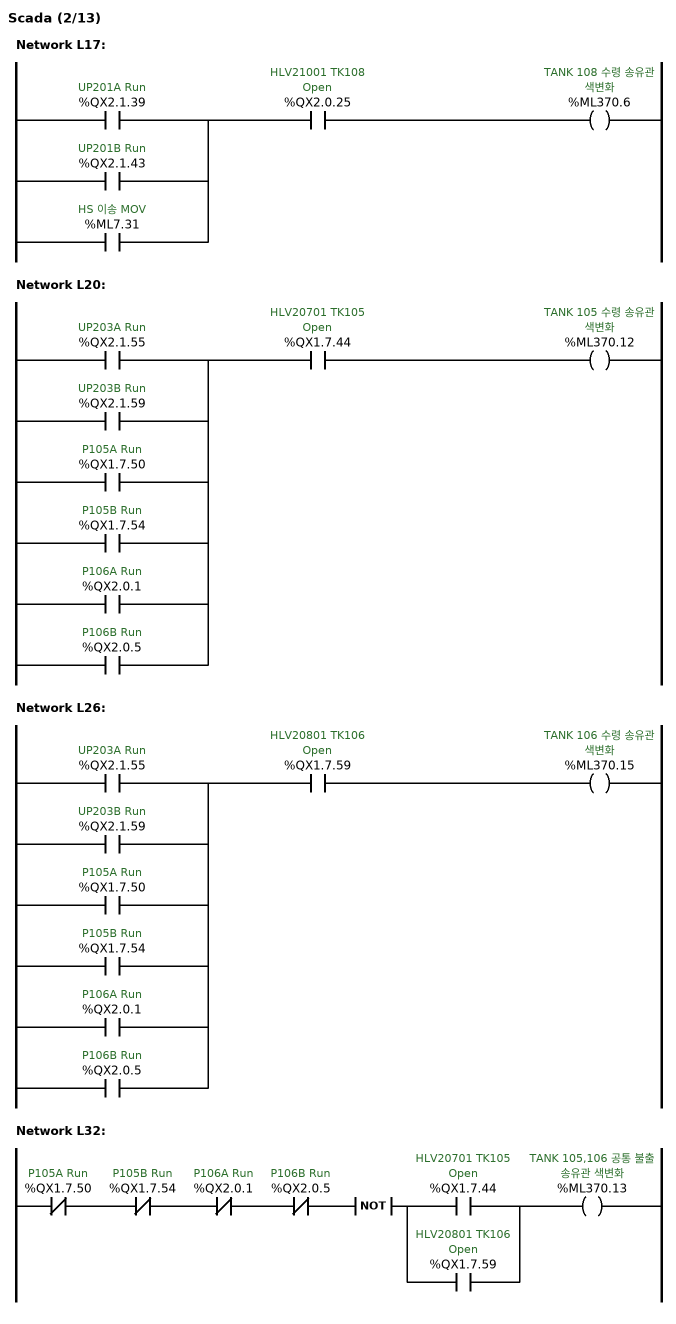
(* [picture p120: Scada rungs L17-L32] *)
(* Rung L17 *)
%ML370.6 := (%QX2.1.39 OR %QX2.1.43 OR %ML7.31) AND %QX2.0.25;
(* Rung L20 *)
%ML370.12 := (%QX2.1.55 OR %QX2.1.59 OR %QX1.7.50 OR %QX1.7.54 OR %QX2.0.1 OR %QX2.0.5) AND %QX1.7.44;
(* Rung L26 *)
%ML370.15 := (%QX2.1.55 OR %QX2.1.59 OR %QX1.7.50 OR %QX1.7.54 OR %QX2.0.1 OR %QX2.0.5) AND %QX1.7.59;
(* Rung L32 *)
%ML370.13 := NOT (NOT %QX1.7.50 AND NOT %QX1.7.54 AND NOT %QX2.0.1 AND NOT %QX2.0.5) AND (%QX1.7.44 OR %QX1.7.59);

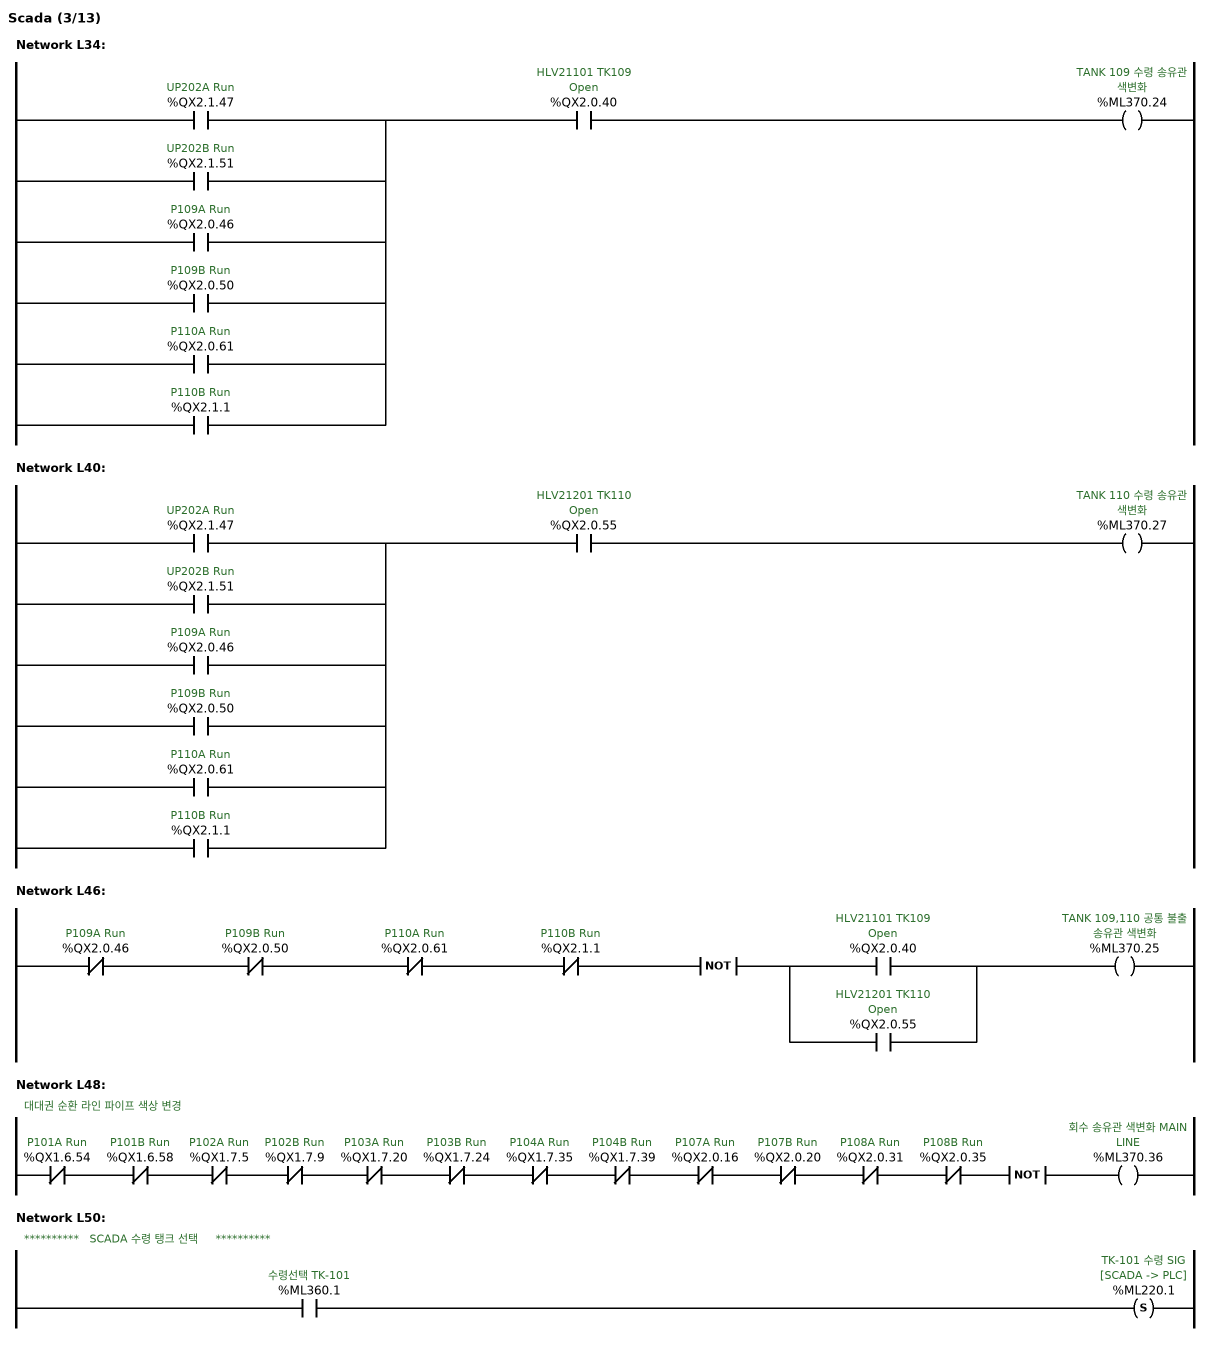
(* Rung L34 *)
%ML370.24 := (%QX2.1.47 OR %QX2.1.51 OR %QX2.0.46 OR %QX2.0.50 OR %QX2.0.61 OR %QX2.1.1) AND %QX2.0.40;
(* Rung L40 *)
%ML370.27 := (%QX2.1.47 OR %QX2.1.51 OR %QX2.0.46 OR %QX2.0.50 OR %QX2.0.61 OR %QX2.1.1) AND %QX2.0.55;
(* Rung L46 *)
%ML370.25 := NOT (NOT %QX2.0.46 AND NOT %QX2.0.50 AND NOT %QX2.0.61 AND NOT %QX2.1.1) AND (%QX2.0.40 OR %QX2.0.55);
(* Rung L48 *)
%ML370.36 := NOT (NOT %QX1.6.54 AND NOT %QX1.6.58 AND NOT %QX1.7.5 AND NOT %QX1.7.9 AND NOT %QX1.7.20 AND NOT %QX1.7.24 AND NOT %QX1.7.35 AND NOT %QX1.7.39 AND NOT %QX2.0.16 AND NOT %QX2.0.20 AND NOT %QX2.0.31 AND NOT %QX2.0.35);
(* 대대권 순환 라인 파이프 색상 변경 *)
(* **********   SCADA 수령 탱크 선택     ********** *)
(* Rung L50 *)
IF %ML360.1 THEN %ML220.1 := TRUE; END_IF;

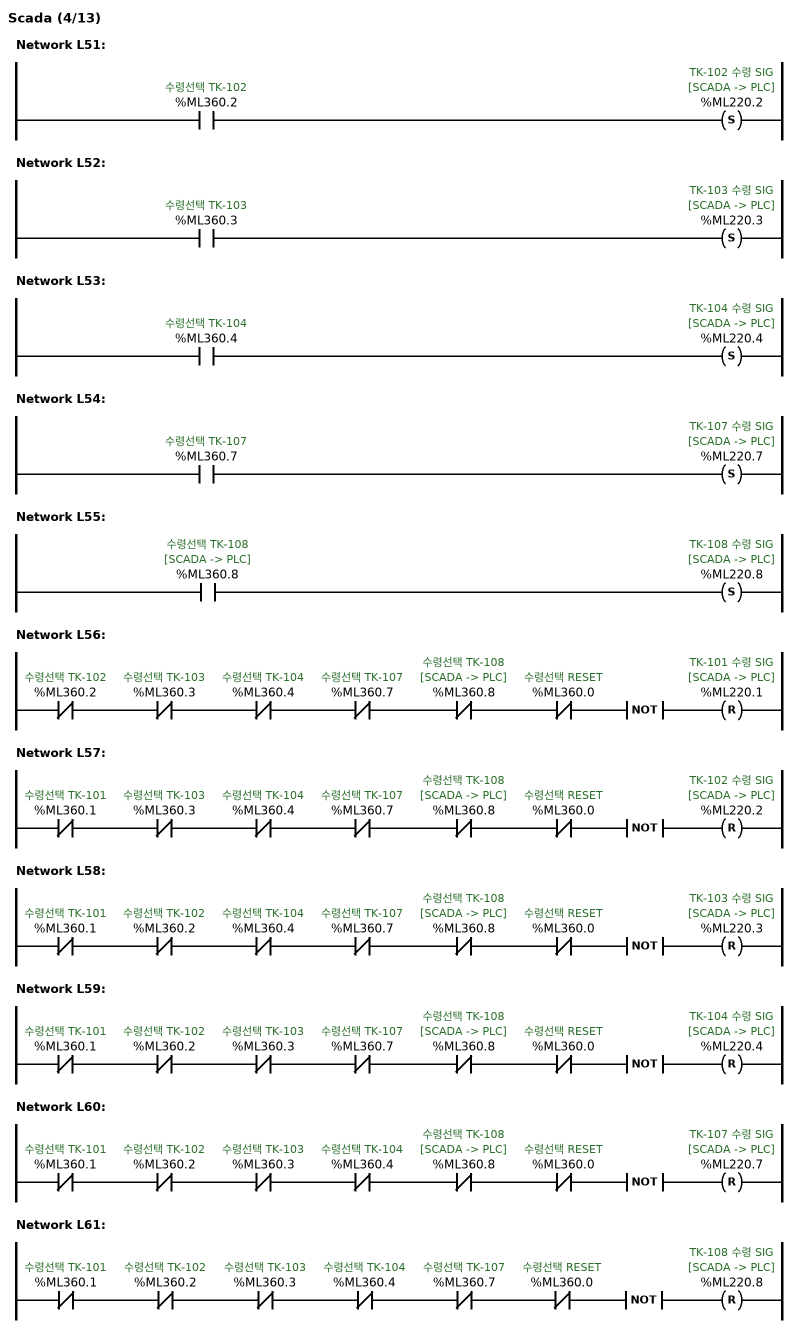
(* Rung L51 *)
IF %ML360.2 THEN %ML220.2 := TRUE; END_IF;
(* Rung L52 *)
IF %ML360.3 THEN %ML220.3 := TRUE; END_IF;
(* Rung L53 *)
IF %ML360.4 THEN %ML220.4 := TRUE; END_IF;
(* Rung L54 *)
IF %ML360.7 THEN %ML220.7 := TRUE; END_IF;
(* Rung L55 *)
IF %ML360.8 THEN %ML220.8 := TRUE; END_IF;
(* Rung L56 *)
IF NOT (NOT %ML360.2 AND NOT %ML360.3 AND NOT %ML360.4 AND NOT %ML360.7 AND NOT %ML360.8 AND NOT %ML360.0) THEN
    %ML220.1 := FALSE;
END_IF;
(* Rung L57 *)
IF NOT (NOT %ML360.1 AND NOT %ML360.3 AND NOT %ML360.4 AND NOT %ML360.7 AND NOT %ML360.8 AND NOT %ML360.0) THEN
    %ML220.2 := FALSE;
END_IF;
(* Rung L58 *)
IF NOT (NOT %ML360.1 AND NOT %ML360.2 AND NOT %ML360.4 AND NOT %ML360.7 AND NOT %ML360.8 AND NOT %ML360.0) THEN
    %ML220.3 := FALSE;
END_IF;
(* Rung L59 *)
IF NOT (NOT %ML360.1 AND NOT %ML360.2 AND NOT %ML360.3 AND NOT %ML360.7 AND NOT %ML360.8 AND NOT %ML360.0) THEN
    %ML220.4 := FALSE;
END_IF;
(* Rung L60 *)
IF NOT (NOT %ML360.1 AND NOT %ML360.2 AND NOT %ML360.3 AND NOT %ML360.4 AND NOT %ML360.8 AND NOT %ML360.0) THEN
    %ML220.7 := FALSE;
END_IF;
(* Rung L61 *)
IF NOT (NOT %ML360.1 AND NOT %ML360.2 AND NOT %ML360.3 AND NOT %ML360.4 AND NOT %ML360.7 AND NOT %ML360.0) THEN
    %ML220.8 := FALSE;
END_IF;

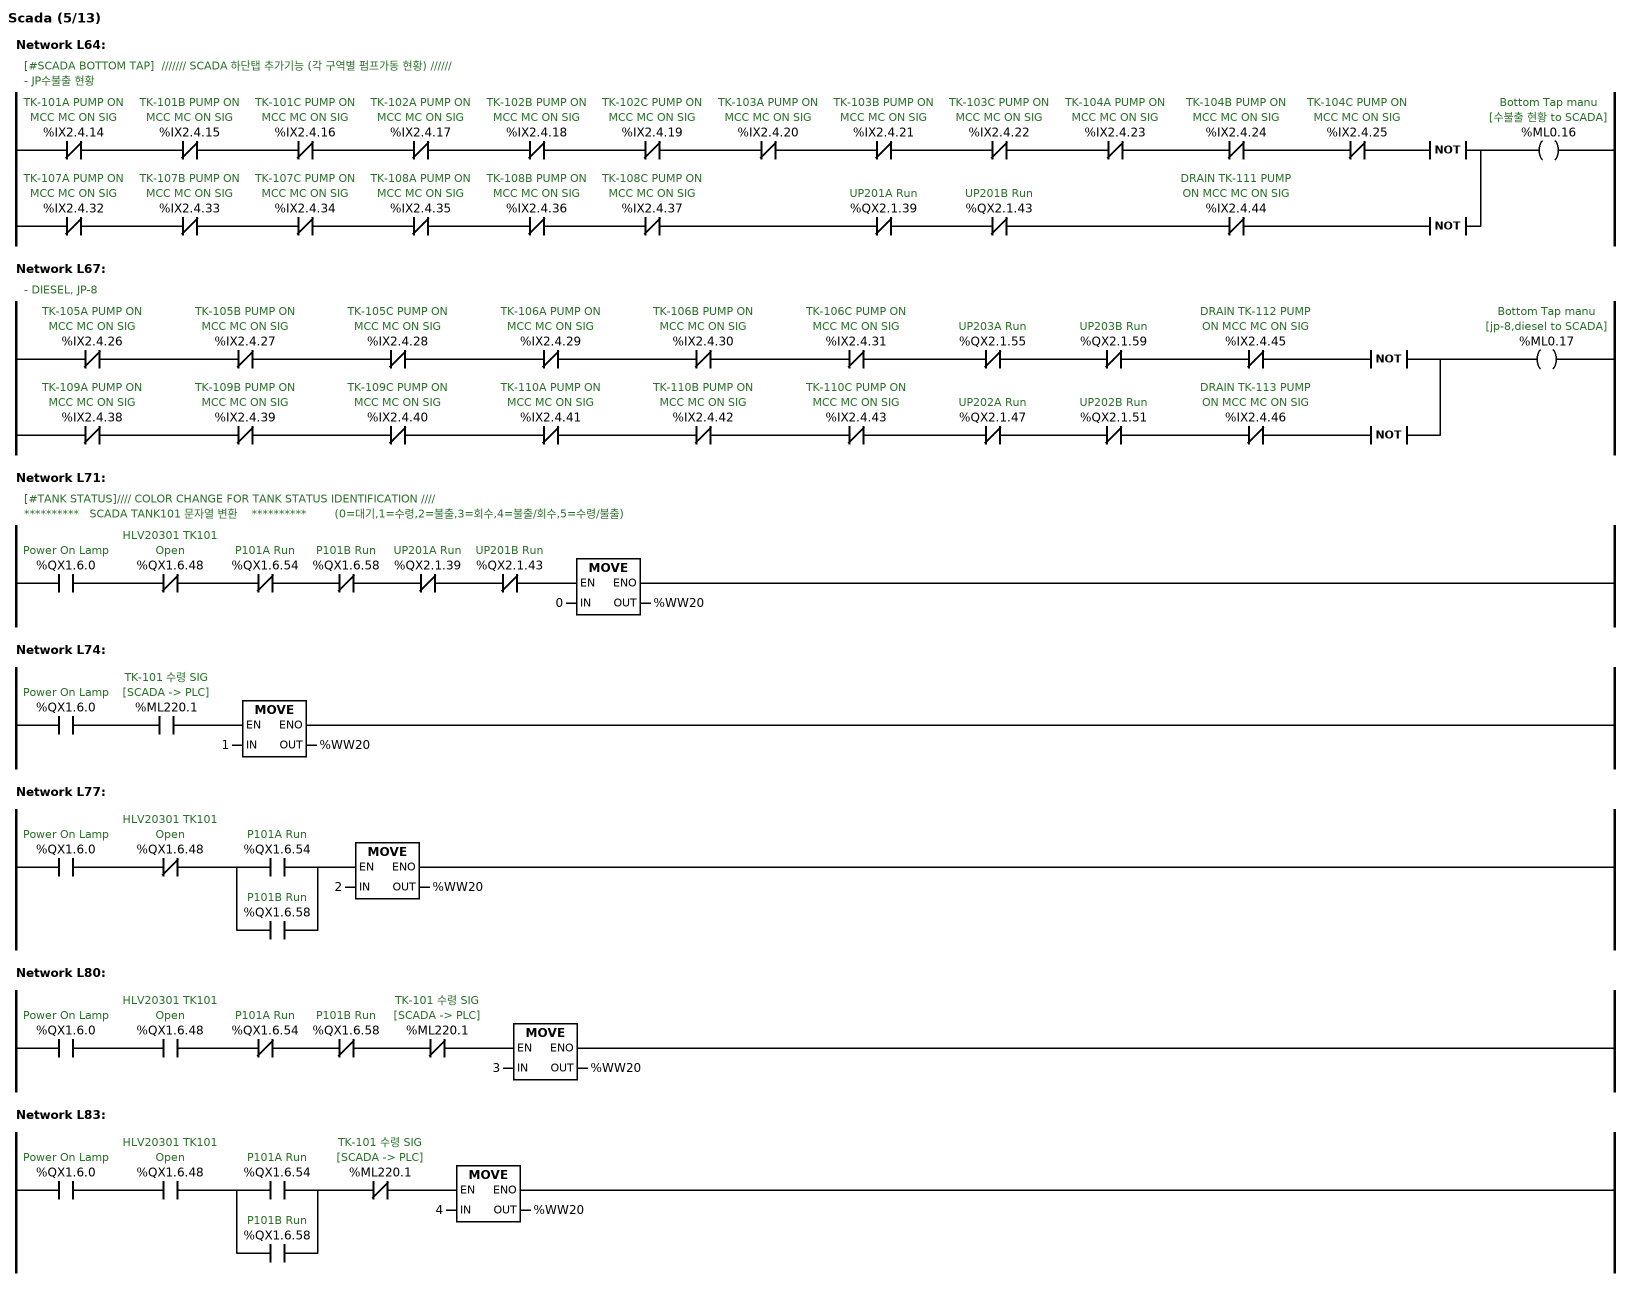
(* [#SCADA BOTTOM TAP]  /////// SCADA 하단탭 추가기능 (각 구역별 펌프가동 현황) ////// *)
(* - JP수불출 현황 *)
(* Rung L64 *)
%ML0.16 := NOT (NOT %IX2.4.14 AND NOT %IX2.4.15 AND NOT %IX2.4.16 AND NOT %IX2.4.17 AND NOT %IX2.4.18 AND NOT %IX2.4.19 AND NOT %IX2.4.20 AND NOT %IX2.4.21 AND NOT %IX2.4.22 AND NOT %IX2.4.23 AND NOT %IX2.4.24 AND NOT %IX2.4.25) OR NOT (NOT %IX2.4.32 AND NOT %IX2.4.33 AND NOT %IX2.4.34 AND NOT %IX2.4.35 AND NOT %IX2.4.36 AND NOT %IX2.4.37 AND NOT %QX2.1.39 AND NOT %QX2.1.43 AND NOT %IX2.4.44);
(* - DIESEL, JP-8 *)
(* Rung L67 *)
%ML0.17 := NOT (NOT %IX2.4.26 AND NOT %IX2.4.27 AND NOT %IX2.4.28 AND NOT %IX2.4.29 AND NOT %IX2.4.30 AND NOT %IX2.4.31 AND NOT %QX2.1.55 AND NOT %QX2.1.59 AND NOT %IX2.4.45) OR NOT (NOT %IX2.4.38 AND NOT %IX2.4.39 AND NOT %IX2.4.40 AND NOT %IX2.4.41 AND NOT %IX2.4.42 AND NOT %IX2.4.43 AND NOT %QX2.1.47 AND NOT %QX2.1.51 AND NOT %IX2.4.46);
(* [#TANK STATUS]//// COLOR CHANGE FOR TANK STATUS IDENTIFICATION //// *)
(* **********   SCADA TANK101 문자열 변환    **********        (0=대기,1=수령,2=불출,3=회수,4=불출/회수,5=수령/불출) *)
(* Rung L71 *)
IF %QX1.6.0 AND NOT %QX1.6.48 AND NOT %QX1.6.54 AND NOT %QX1.6.58 AND NOT %QX2.1.39 AND NOT %QX2.1.43 THEN
    %WW20 := 0;
END_IF;
(* Rung L74 *)
IF %QX1.6.0 AND %ML220.1 THEN %WW20 := 1; END_IF;
(* Rung L77 *)
IF %QX1.6.0 AND NOT %QX1.6.48 AND (%QX1.6.54 OR %QX1.6.58) THEN %WW20 := 2; END_IF;
(* Rung L80 *)
IF %QX1.6.0 AND %QX1.6.48 AND NOT %QX1.6.54 AND NOT %QX1.6.58 AND NOT %ML220.1 THEN %WW20 := 3; END_IF;
(* Rung L83 *)
IF %QX1.6.0 AND %QX1.6.48 AND (%QX1.6.54 OR %QX1.6.58) AND NOT %ML220.1 THEN %WW20 := 4; END_IF;

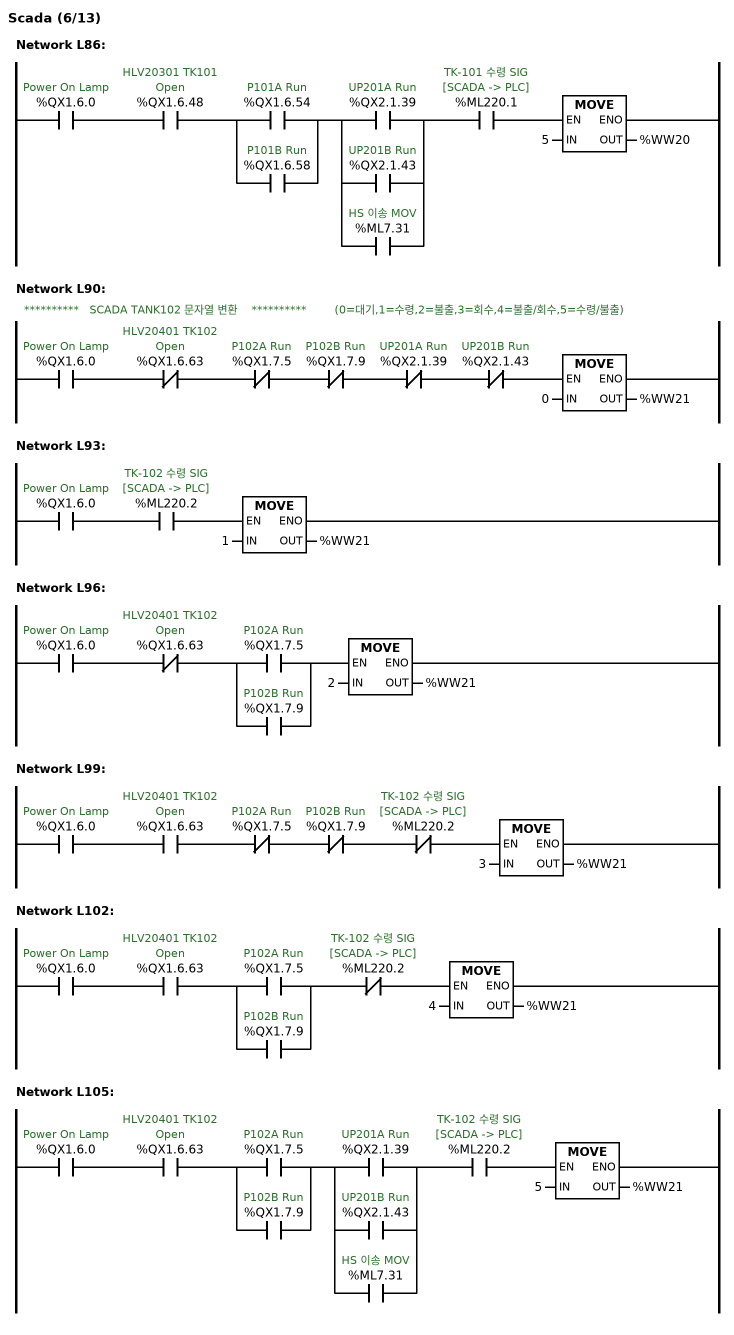
(* Rung L86 *)
IF %QX1.6.0 AND %QX1.6.48 AND (%QX1.6.54 OR %QX1.6.58) AND (%QX2.1.39 OR %QX2.1.43 OR %ML7.31) AND %ML220.1 THEN
    %WW20 := 5;
END_IF;
(* **********   SCADA TANK102 문자열 변환    **********        (0=대기,1=수령,2=불출,3=회수,4=불출/회수,5=수령/불출) *)
(* Rung L90 *)
IF %QX1.6.0 AND NOT %QX1.6.63 AND NOT %QX1.7.5 AND NOT %QX1.7.9 AND NOT %QX2.1.39 AND NOT %QX2.1.43 THEN
    %WW21 := 0;
END_IF;
(* Rung L93 *)
IF %QX1.6.0 AND %ML220.2 THEN %WW21 := 1; END_IF;
(* Rung L96 *)
IF %QX1.6.0 AND NOT %QX1.6.63 AND (%QX1.7.5 OR %QX1.7.9) THEN %WW21 := 2; END_IF;
(* Rung L99 *)
IF %QX1.6.0 AND %QX1.6.63 AND NOT %QX1.7.5 AND NOT %QX1.7.9 AND NOT %ML220.2 THEN %WW21 := 3; END_IF;
(* Rung L102 *)
IF %QX1.6.0 AND %QX1.6.63 AND (%QX1.7.5 OR %QX1.7.9) AND NOT %ML220.2 THEN %WW21 := 4; END_IF;
(* Rung L105 *)
IF %QX1.6.0 AND %QX1.6.63 AND (%QX1.7.5 OR %QX1.7.9) AND (%QX2.1.39 OR %QX2.1.43 OR %ML7.31) AND %ML220.2 THEN
    %WW21 := 5;
END_IF;

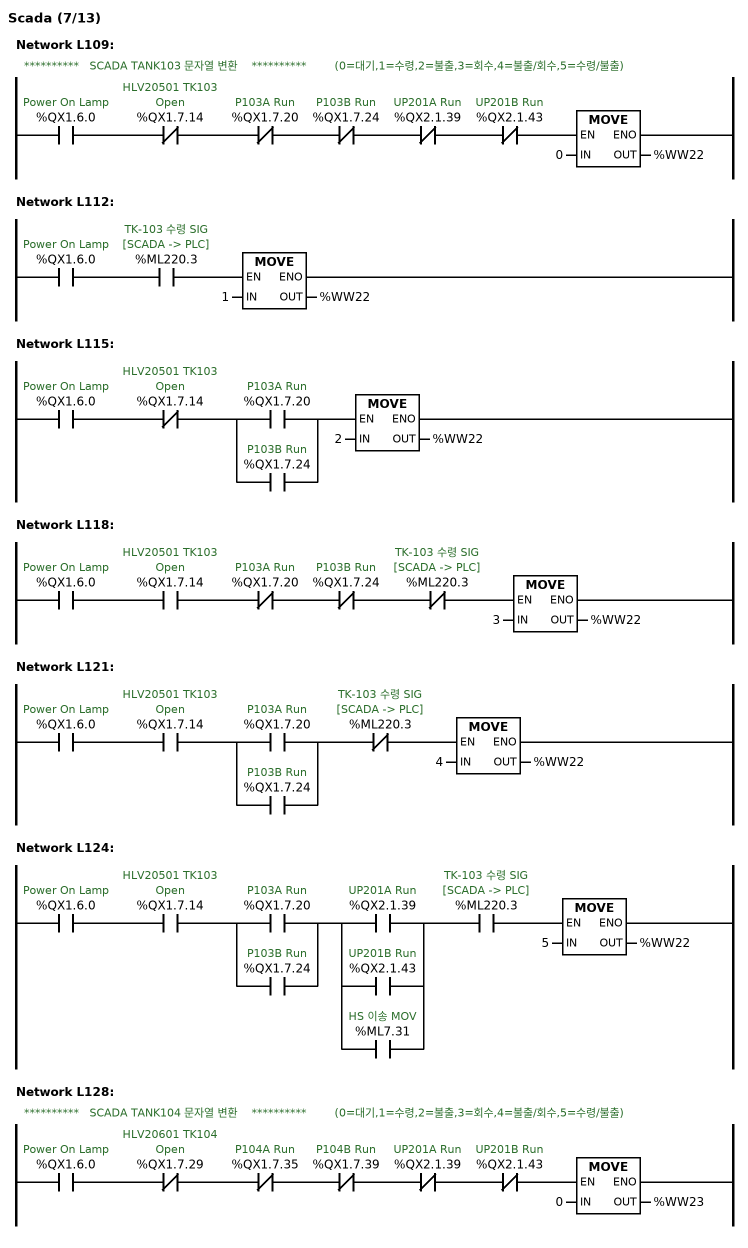
(* **********   SCADA TANK103 문자열 변환    **********        (0=대기,1=수령,2=불출,3=회수,4=불출/회수,5=수령/불출) *)
(* Rung L109 *)
IF %QX1.6.0 AND NOT %QX1.7.14 AND NOT %QX1.7.20 AND NOT %QX1.7.24 AND NOT %QX2.1.39 AND NOT %QX2.1.43 THEN
    %WW22 := 0;
END_IF;
(* Rung L112 *)
IF %QX1.6.0 AND %ML220.3 THEN %WW22 := 1; END_IF;
(* Rung L115 *)
IF %QX1.6.0 AND NOT %QX1.7.14 AND (%QX1.7.20 OR %QX1.7.24) THEN %WW22 := 2; END_IF;
(* Rung L118 *)
IF %QX1.6.0 AND %QX1.7.14 AND NOT %QX1.7.20 AND NOT %QX1.7.24 AND NOT %ML220.3 THEN %WW22 := 3; END_IF;
(* Rung L121 *)
IF %QX1.6.0 AND %QX1.7.14 AND (%QX1.7.20 OR %QX1.7.24) AND NOT %ML220.3 THEN %WW22 := 4; END_IF;
(* Rung L124 *)
IF %QX1.6.0 AND %QX1.7.14 AND (%QX1.7.20 OR %QX1.7.24) AND (%QX2.1.39 OR %QX2.1.43 OR %ML7.31) AND %ML220.3 THEN
    %WW22 := 5;
END_IF;
(* **********   SCADA TANK104 문자열 변환    **********        (0=대기,1=수령,2=불출,3=회수,4=불출/회수,5=수령/불출) *)
(* Rung L128 *)
IF %QX1.6.0 AND NOT %QX1.7.29 AND NOT %QX1.7.35 AND NOT %QX1.7.39 AND NOT %QX2.1.39 AND NOT %QX2.1.43 THEN
    %WW23 := 0;
END_IF;

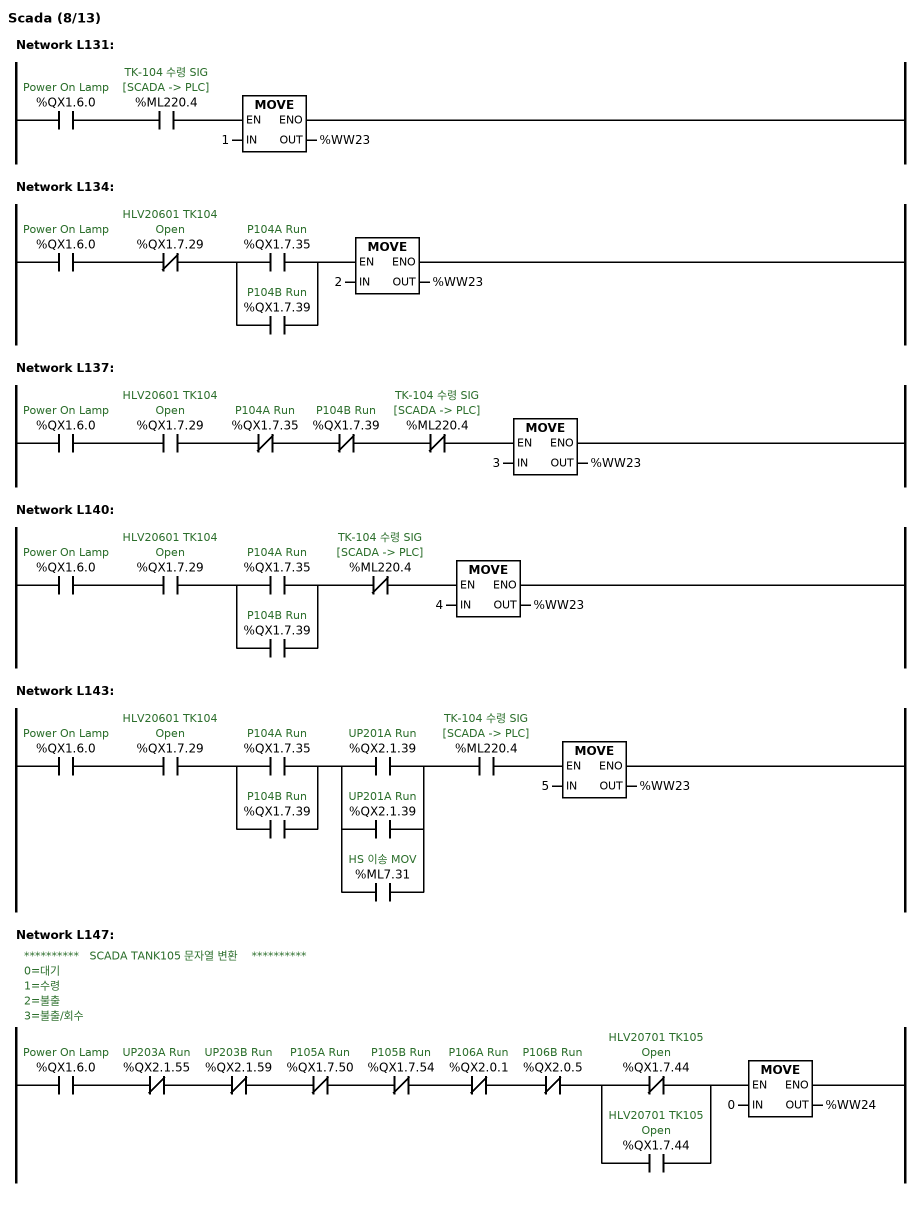
(* Rung L131 *)
IF %QX1.6.0 AND %ML220.4 THEN %WW23 := 1; END_IF;
(* Rung L134 *)
IF %QX1.6.0 AND NOT %QX1.7.29 AND (%QX1.7.35 OR %QX1.7.39) THEN %WW23 := 2; END_IF;
(* Rung L137 *)
IF %QX1.6.0 AND %QX1.7.29 AND NOT %QX1.7.35 AND NOT %QX1.7.39 AND NOT %ML220.4 THEN %WW23 := 3; END_IF;
(* Rung L140 *)
IF %QX1.6.0 AND %QX1.7.29 AND (%QX1.7.35 OR %QX1.7.39) AND NOT %ML220.4 THEN %WW23 := 4; END_IF;
(* Rung L143 *)
IF %QX1.6.0 AND %QX1.7.29 AND (%QX1.7.35 OR %QX1.7.39) AND (%QX2.1.39 OR %QX2.1.39 OR %ML7.31) AND %ML220.4 THEN
    %WW23 := 5;
END_IF;
(* **********   SCADA TANK105 문자열 변환    ********** / 0=대기 / 1=수령 / 2=불출 / 3=불출/회수 *)
(* Rung L147 *)
IF %QX1.6.0 AND NOT %QX2.1.55 AND NOT %QX2.1.59 AND NOT %QX1.7.50 AND NOT %QX1.7.54 AND NOT %QX2.0.1 AND NOT %QX2.0.5 AND (NOT %QX1.7.44 OR %QX1.7.44) THEN
    %WW24 := 0;
END_IF;

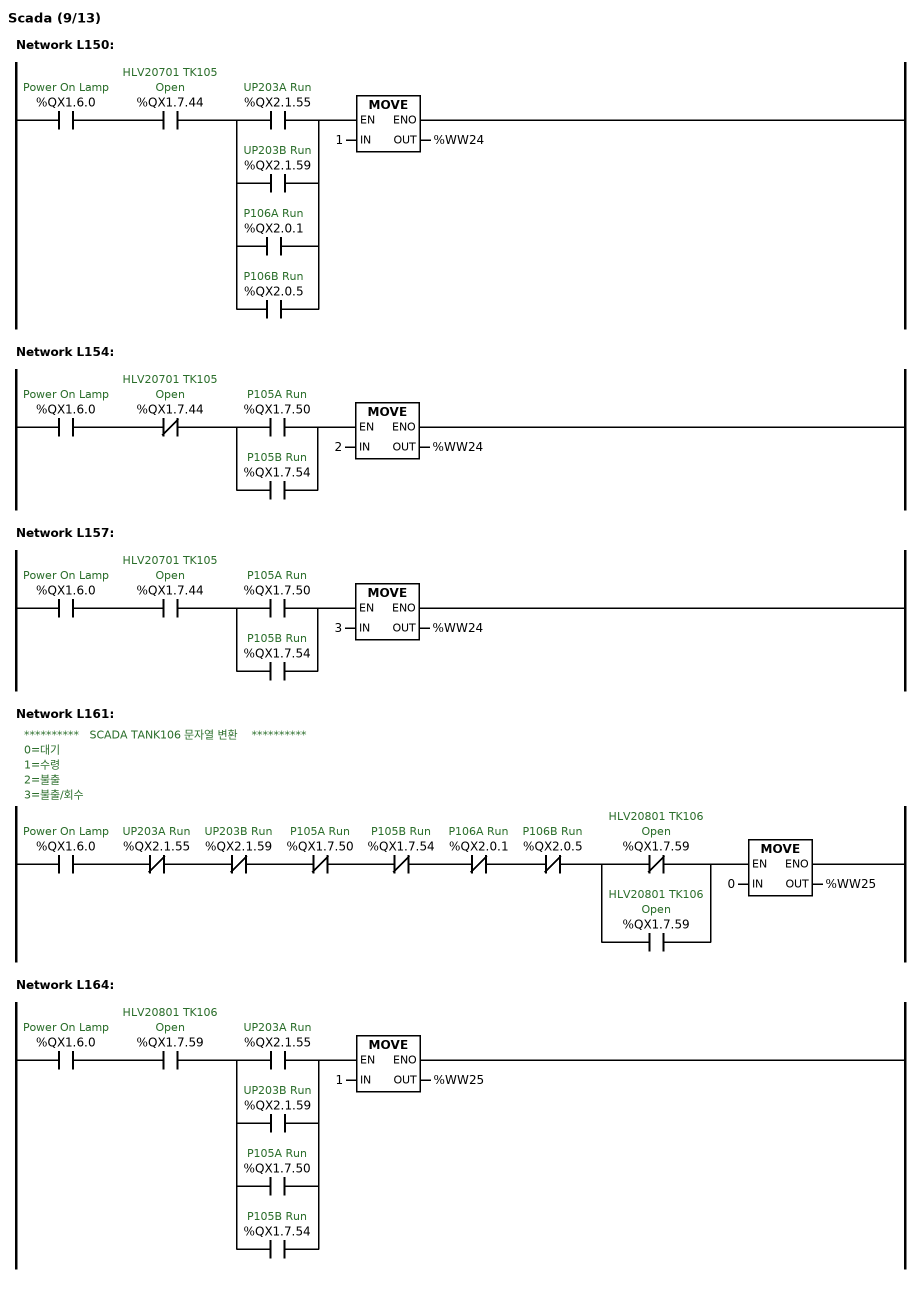
(* Rung L150 *)
IF %QX1.6.0 AND %QX1.7.44 AND (%QX2.1.55 OR %QX2.1.59 OR %QX2.0.1 OR %QX2.0.5) THEN %WW24 := 1; END_IF;
(* Rung L154 *)
IF %QX1.6.0 AND NOT %QX1.7.44 AND (%QX1.7.50 OR %QX1.7.54) THEN %WW24 := 2; END_IF;
(* Rung L157 *)
IF %QX1.6.0 AND %QX1.7.44 AND (%QX1.7.50 OR %QX1.7.54) THEN %WW24 := 3; END_IF;
(* **********   SCADA TANK106 문자열 변환    ********** / 0=대기 / 1=수령 / 2=불출 / 3=불출/회수 *)
(* Rung L161 *)
IF %QX1.6.0 AND NOT %QX2.1.55 AND NOT %QX2.1.59 AND NOT %QX1.7.50 AND NOT %QX1.7.54 AND NOT %QX2.0.1 AND NOT %QX2.0.5 AND (NOT %QX1.7.59 OR %QX1.7.59) THEN
    %WW25 := 0;
END_IF;
(* Rung L164 *)
IF %QX1.6.0 AND %QX1.7.59 AND (%QX2.1.55 OR %QX2.1.59 OR %QX1.7.50 OR %QX1.7.54) THEN %WW25 := 1; END_IF;

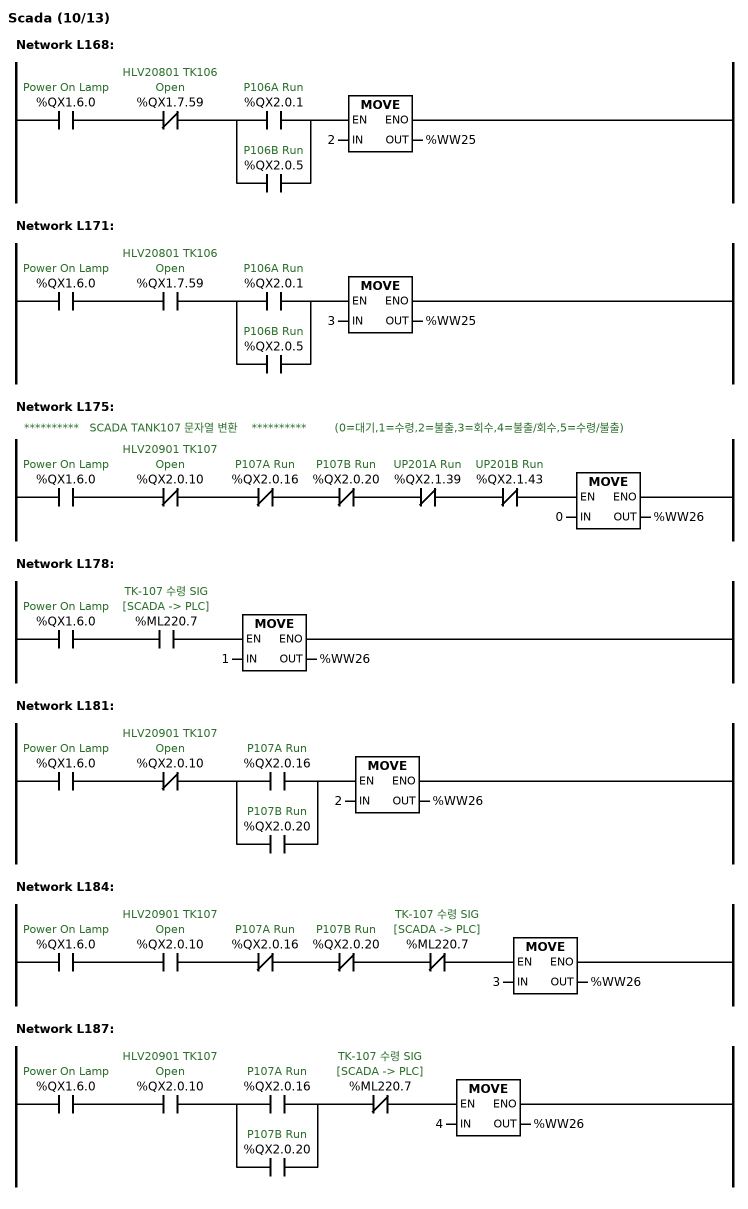
(* Rung L168 *)
IF %QX1.6.0 AND NOT %QX1.7.59 AND (%QX2.0.1 OR %QX2.0.5) THEN %WW25 := 2; END_IF;
(* Rung L171 *)
IF %QX1.6.0 AND %QX1.7.59 AND (%QX2.0.1 OR %QX2.0.5) THEN %WW25 := 3; END_IF;
(* **********   SCADA TANK107 문자열 변환    **********        (0=대기,1=수령,2=불출,3=회수,4=불출/회수,5=수령/불출) *)
(* Rung L175 *)
IF %QX1.6.0 AND NOT %QX2.0.10 AND NOT %QX2.0.16 AND NOT %QX2.0.20 AND NOT %QX2.1.39 AND NOT %QX2.1.43 THEN
    %WW26 := 0;
END_IF;
(* Rung L178 *)
IF %QX1.6.0 AND %ML220.7 THEN %WW26 := 1; END_IF;
(* Rung L181 *)
IF %QX1.6.0 AND NOT %QX2.0.10 AND (%QX2.0.16 OR %QX2.0.20) THEN %WW26 := 2; END_IF;
(* Rung L184 *)
IF %QX1.6.0 AND %QX2.0.10 AND NOT %QX2.0.16 AND NOT %QX2.0.20 AND NOT %ML220.7 THEN %WW26 := 3; END_IF;
(* Rung L187 *)
IF %QX1.6.0 AND %QX2.0.10 AND (%QX2.0.16 OR %QX2.0.20) AND NOT %ML220.7 THEN %WW26 := 4; END_IF;

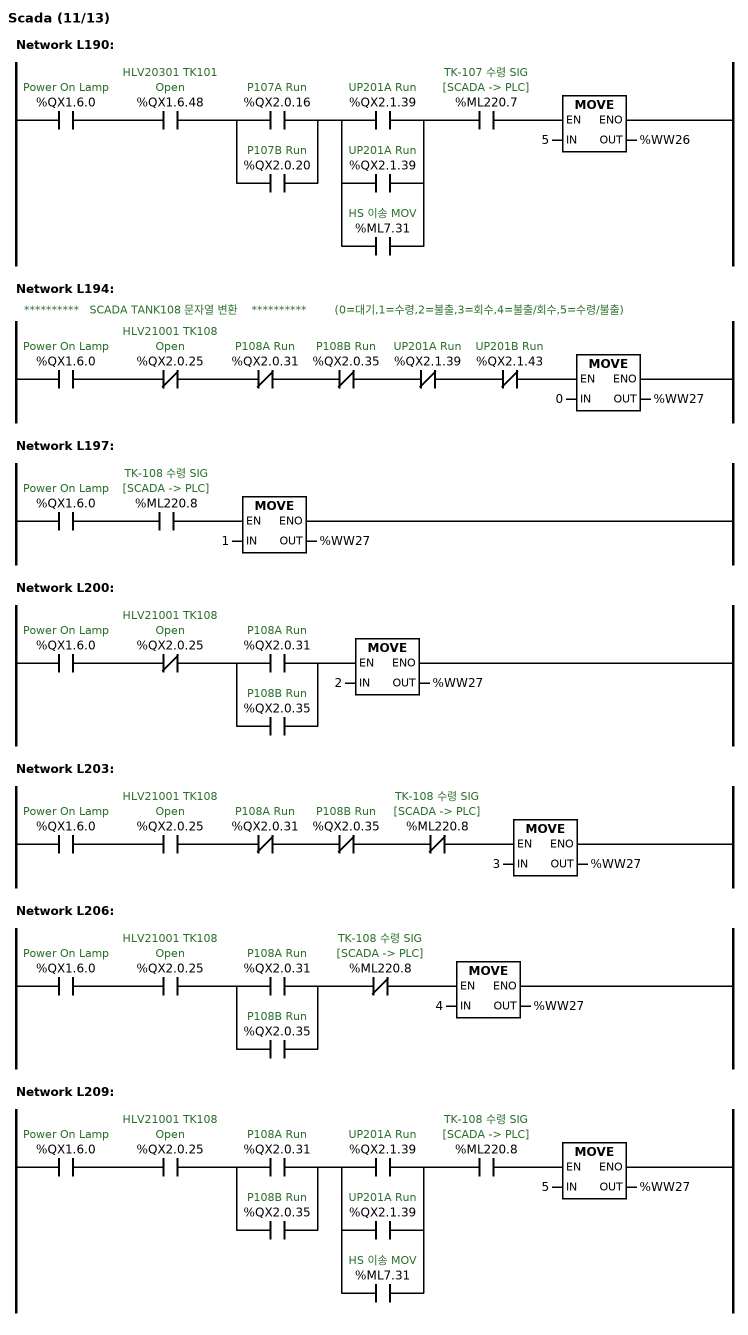
(* Rung L190 *)
IF %QX1.6.0 AND %QX1.6.48 AND (%QX2.0.16 OR %QX2.0.20) AND (%QX2.1.39 OR %QX2.1.39 OR %ML7.31) AND %ML220.7 THEN
    %WW26 := 5;
END_IF;
(* **********   SCADA TANK108 문자열 변환    **********        (0=대기,1=수령,2=불출,3=회수,4=불출/회수,5=수령/불출) *)
(* Rung L194 *)
IF %QX1.6.0 AND NOT %QX2.0.25 AND NOT %QX2.0.31 AND NOT %QX2.0.35 AND NOT %QX2.1.39 AND NOT %QX2.1.43 THEN
    %WW27 := 0;
END_IF;
(* Rung L197 *)
IF %QX1.6.0 AND %ML220.8 THEN %WW27 := 1; END_IF;
(* Rung L200 *)
IF %QX1.6.0 AND NOT %QX2.0.25 AND (%QX2.0.31 OR %QX2.0.35) THEN %WW27 := 2; END_IF;
(* Rung L203 *)
IF %QX1.6.0 AND %QX2.0.25 AND NOT %QX2.0.31 AND NOT %QX2.0.35 AND NOT %ML220.8 THEN %WW27 := 3; END_IF;
(* Rung L206 *)
IF %QX1.6.0 AND %QX2.0.25 AND (%QX2.0.31 OR %QX2.0.35) AND NOT %ML220.8 THEN %WW27 := 4; END_IF;
(* Rung L209 *)
IF %QX1.6.0 AND %QX2.0.25 AND (%QX2.0.31 OR %QX2.0.35) AND (%QX2.1.39 OR %QX2.1.39 OR %ML7.31) AND %ML220.8 THEN
    %WW27 := 5;
END_IF;

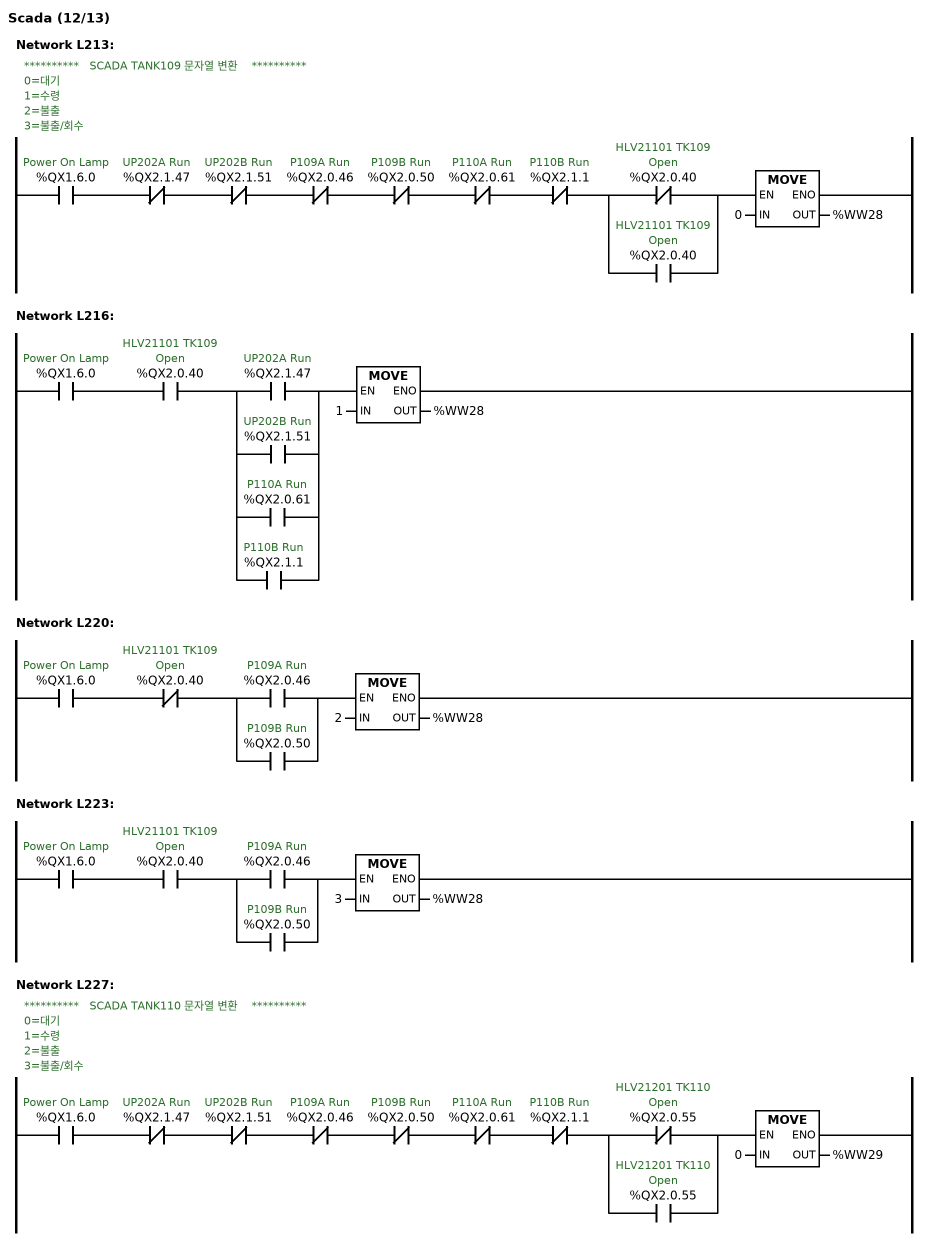
(* **********   SCADA TANK109 문자열 변환    ********** / 0=대기 / 1=수령 / 2=불출 / 3=불출/회수 *)
(* Rung L213 *)
IF %QX1.6.0 AND NOT %QX2.1.47 AND NOT %QX2.1.51 AND NOT %QX2.0.46 AND NOT %QX2.0.50 AND NOT %QX2.0.61 AND NOT %QX2.1.1 AND (NOT %QX2.0.40 OR %QX2.0.40) THEN
    %WW28 := 0;
END_IF;
(* Rung L216 *)
IF %QX1.6.0 AND %QX2.0.40 AND (%QX2.1.47 OR %QX2.1.51 OR %QX2.0.61 OR %QX2.1.1) THEN %WW28 := 1; END_IF;
(* Rung L220 *)
IF %QX1.6.0 AND NOT %QX2.0.40 AND (%QX2.0.46 OR %QX2.0.50) THEN %WW28 := 2; END_IF;
(* Rung L223 *)
IF %QX1.6.0 AND %QX2.0.40 AND (%QX2.0.46 OR %QX2.0.50) THEN %WW28 := 3; END_IF;
(* **********   SCADA TANK110 문자열 변환    ********** / 0=대기 / 1=수령 / 2=불출 / 3=불출/회수 *)
(* Rung L227 *)
IF %QX1.6.0 AND NOT %QX2.1.47 AND NOT %QX2.1.51 AND NOT %QX2.0.46 AND NOT %QX2.0.50 AND NOT %QX2.0.61 AND NOT %QX2.1.1 AND (NOT %QX2.0.55 OR %QX2.0.55) THEN
    %WW29 := 0;
END_IF;

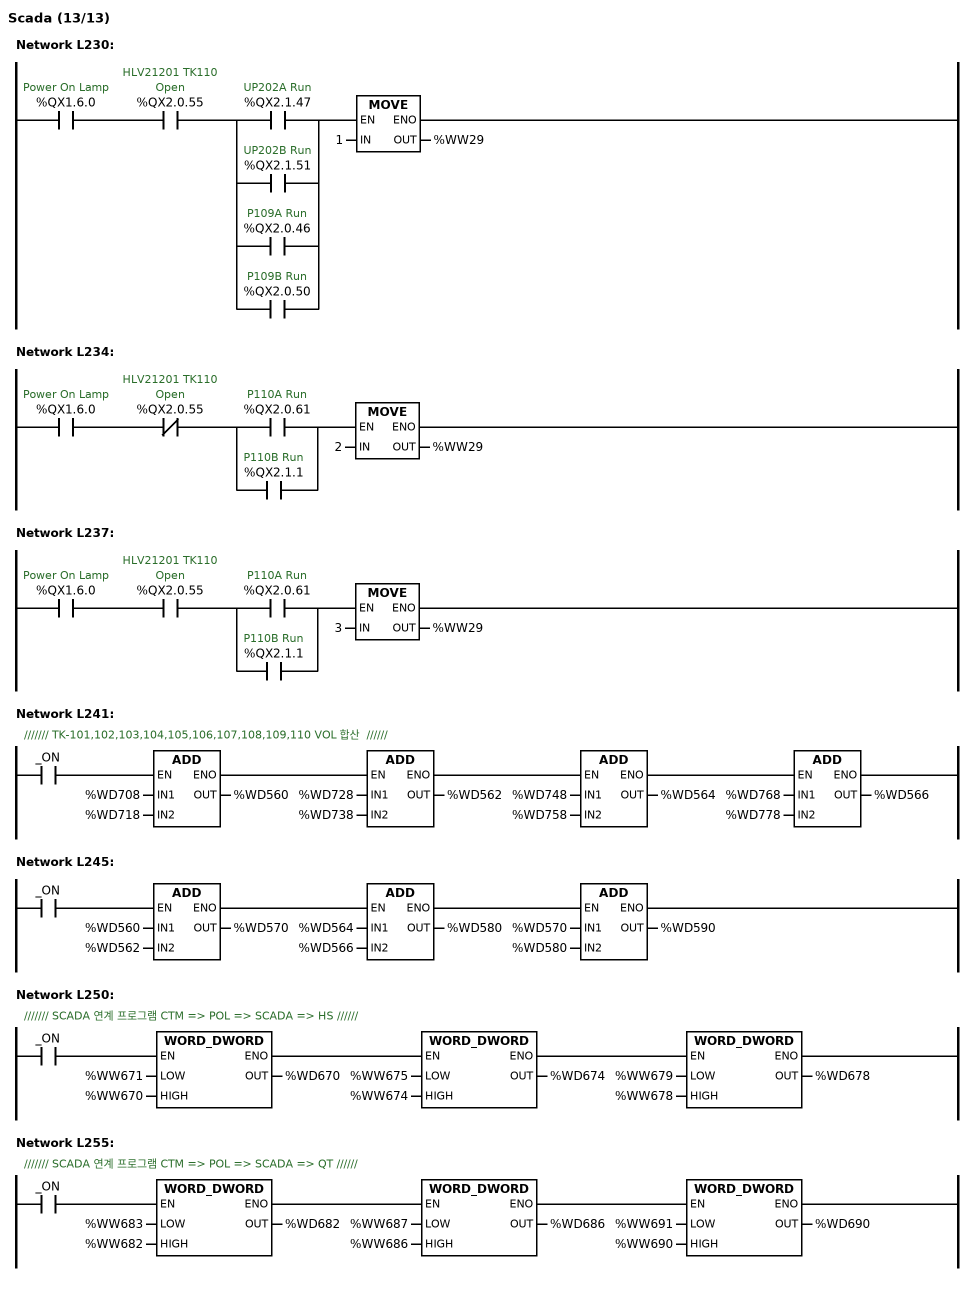
(* Rung L230 *)
IF %QX1.6.0 AND %QX2.0.55 AND (%QX2.1.47 OR %QX2.1.51 OR %QX2.0.46 OR %QX2.0.50) THEN %WW29 := 1; END_IF;
(* Rung L234 *)
IF %QX1.6.0 AND NOT %QX2.0.55 AND (%QX2.0.61 OR %QX2.1.1) THEN %WW29 := 2; END_IF;
(* Rung L237 *)
IF %QX1.6.0 AND %QX2.0.55 AND (%QX2.0.61 OR %QX2.1.1) THEN %WW29 := 3; END_IF;
(* /////// TK-101,102,103,104,105,106,107,108,109,110 VOL 합산  ////// *)
(* Rung L241 *)
IF _ON THEN
    %WD560 := %WD708 + %WD718;
    %WD562 := %WD728 + %WD738;
    %WD564 := %WD748 + %WD758;
    %WD566 := %WD768 + %WD778;
END_IF;
(* Rung L245 *)
IF _ON THEN
    %WD570 := %WD560 + %WD562;
    %WD580 := %WD564 + %WD566;
    %WD590 := %WD570 + %WD580;
END_IF;
(* /////// SCADA 연계 프로그램 CTM => POL => SCADA => HS ////// *)
(* Rung L250 *)
IF _ON THEN
    %WD670 := WORD_DWORD(LOW := %WW671, HIGH := %WW670);
    %WD674 := WORD_DWORD(LOW := %WW675, HIGH := %WW674);
    %WD678 := WORD_DWORD(LOW := %WW679, HIGH := %WW678);
END_IF;
(* /////// SCADA 연계 프로그램 CTM => POL => SCADA => QT ////// *)
(* Rung L255 *)
IF _ON THEN
    %WD682 := WORD_DWORD(LOW := %WW683, HIGH := %WW682);
    %WD686 := WORD_DWORD(LOW := %WW687, HIGH := %WW686);
    %WD690 := WORD_DWORD(LOW := %WW691, HIGH := %WW690);
END_IF;
END_PROGRAM

PROGRAM Setting (* task: 스캔 프로그램 *)
VAR
    HLV_TK101_PANEL : FF;
    HLV_TK102_PANEL : FF;
    HLV_TK103_PANEL : FF;
    HLV_TK104_PANEL : FF;
    HLV_TK105_PANEL : FF;
    HLV_TK106_PANEL : FF;
    HLV_TK107_PANEL : FF;
    HLV_TK108_PANEL : FF;
    HLV_TK109_PANEL : FF;
    HLV_TK110_PANEL : FF;
    INST : FF;
END_VAR
VAR
    _t1 : BOOL;
    _t2 : BOOL;
    _t3 : BOOL;
    _t4 : BOOL;
    _t5 : BOOL;
    _t6 : BOOL;
    _e7 : R_TRIG;
    _e8 : R_TRIG;
    _e9 : R_TRIG;
    _e10 : R_TRIG;
    _t11 : BOOL;
    _t12 : BOOL;
    _t13 : BOOL;
    _t14 : BOOL;
    _t15 : BOOL;
    _t16 : BOOL;
    _t17 : BOOL;
    _t18 : BOOL;
    _t19 : BOOL;
    _t20 : BOOL;
    _t21 : BOOL;
    _t22 : BOOL;
    _t23 : BOOL;
    _t24 : BOOL;
    _t25 : BOOL;
    _t26 : BOOL;
    _t27 : BOOL;
    _t28 : BOOL;
    _t29 : BOOL;
    _t30 : BOOL;
    _t31 : BOOL;
    _t32 : BOOL;
    _t33 : BOOL;
    _t34 : BOOL;
END_VAR

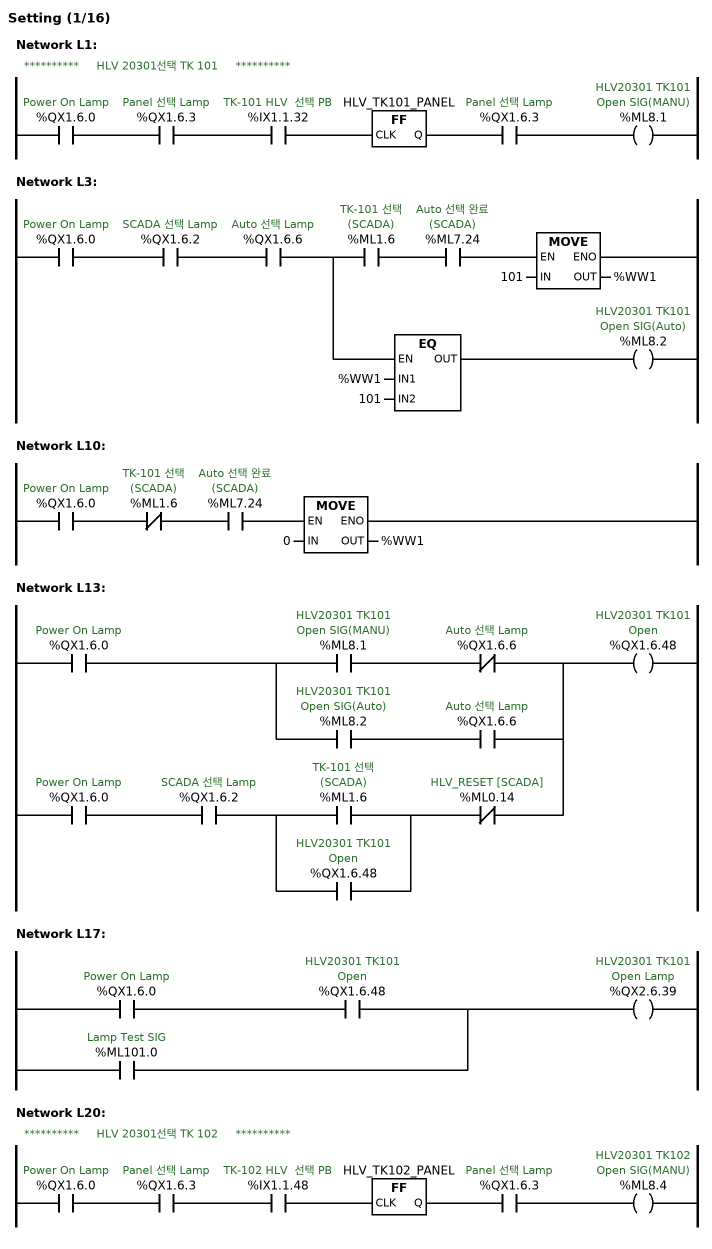
(* **********     HLV 20301선택 TK 101     ********** *)
(* Rung L1 *)
HLV_TK101_PANEL(CLK := %QX1.6.0 AND %QX1.6.3 AND %IX1.1.32);
%ML8.1 := HLV_TK101_PANEL.Q AND %QX1.6.3;
(* Rung L3 *)
IF %QX1.6.0 AND %QX1.6.2 AND %QX1.6.6 AND %ML1.6 AND %ML7.24 THEN %WW1 := 101; END_IF;
IF %QX1.6.0 AND %QX1.6.2 AND %QX1.6.6 THEN _t1 := %WW1 = 101; END_IF;
%ML8.2 := _t1;
(* Rung L10 *)
IF %QX1.6.0 AND NOT %ML1.6 AND %ML7.24 THEN %WW1 := 0; END_IF;
(* Rung L13 *)
%QX1.6.48 := (%QX1.6.0 AND ((%ML8.1 AND NOT %QX1.6.6) OR (%ML8.2 AND %QX1.6.6))) OR (%QX1.6.0 AND %QX1.6.2 AND (%ML1.6 OR %QX1.6.48) AND NOT %ML0.14);
(* Rung L17 *)
%QX2.6.39 := (%QX1.6.0 AND %QX1.6.48) OR %ML101.0;
(* **********     HLV 20301선택 TK 102     ********** *)
(* Rung L20 *)
HLV_TK102_PANEL(CLK := %QX1.6.0 AND %QX1.6.3 AND %IX1.1.48);
%ML8.4 := HLV_TK102_PANEL.Q AND %QX1.6.3;

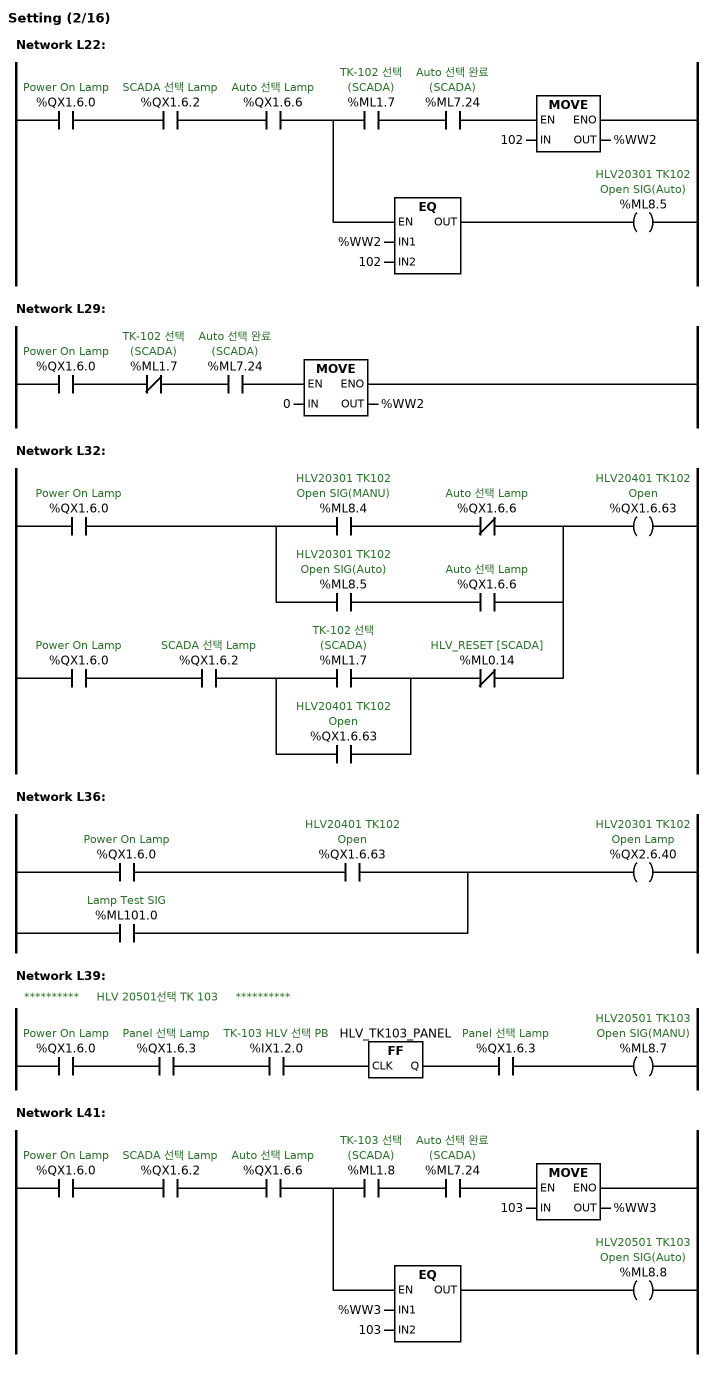
(* Rung L22 *)
IF %QX1.6.0 AND %QX1.6.2 AND %QX1.6.6 AND %ML1.7 AND %ML7.24 THEN %WW2 := 102; END_IF;
IF %QX1.6.0 AND %QX1.6.2 AND %QX1.6.6 THEN _t2 := %WW2 = 102; END_IF;
%ML8.5 := _t2;
(* Rung L29 *)
IF %QX1.6.0 AND NOT %ML1.7 AND %ML7.24 THEN %WW2 := 0; END_IF;
(* Rung L32 *)
%QX1.6.63 := (%QX1.6.0 AND ((%ML8.4 AND NOT %QX1.6.6) OR (%ML8.5 AND %QX1.6.6))) OR (%QX1.6.0 AND %QX1.6.2 AND (%ML1.7 OR %QX1.6.63) AND NOT %ML0.14);
(* Rung L36 *)
%QX2.6.40 := (%QX1.6.0 AND %QX1.6.63) OR %ML101.0;
(* **********     HLV 20501선택 TK 103     ********** *)
(* Rung L39 *)
HLV_TK103_PANEL(CLK := %QX1.6.0 AND %QX1.6.3 AND %IX1.2.0);
%ML8.7 := HLV_TK103_PANEL.Q AND %QX1.6.3;
(* Rung L41 *)
IF %QX1.6.0 AND %QX1.6.2 AND %QX1.6.6 AND %ML1.8 AND %ML7.24 THEN %WW3 := 103; END_IF;
IF %QX1.6.0 AND %QX1.6.2 AND %QX1.6.6 THEN _t3 := %WW3 = 103; END_IF;
%ML8.8 := _t3;

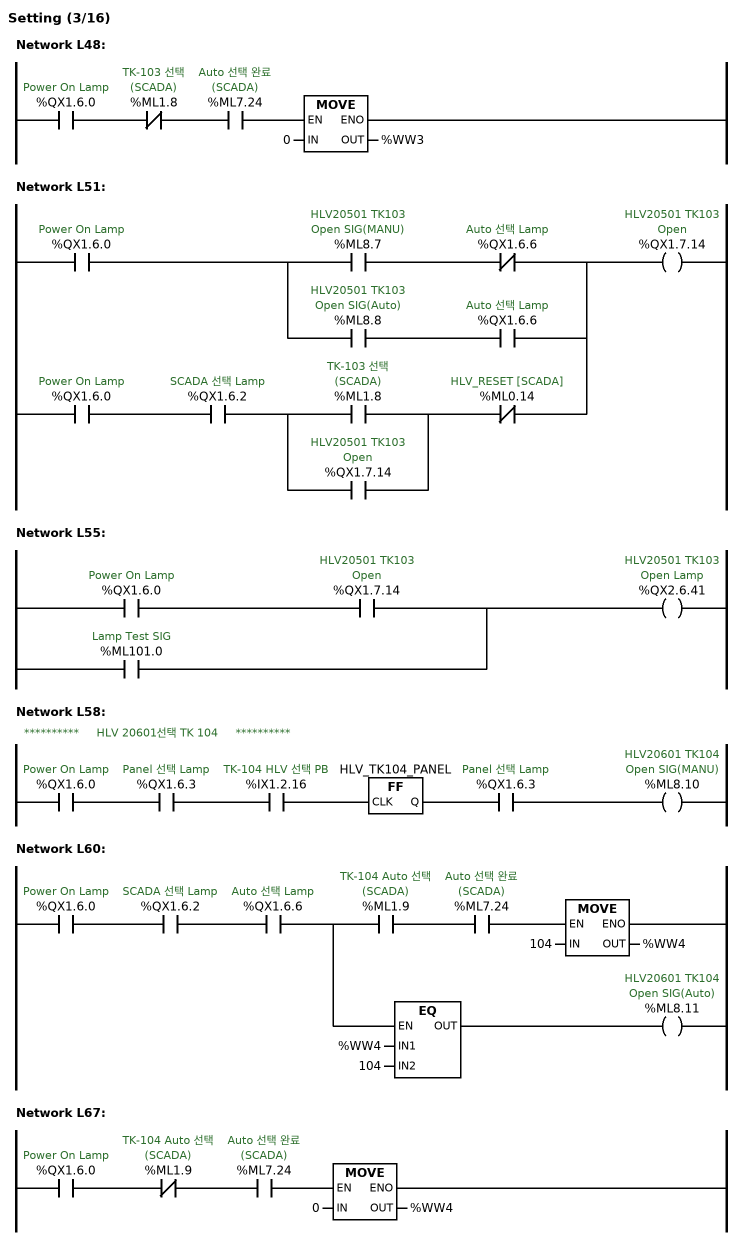
(* Rung L48 *)
IF %QX1.6.0 AND NOT %ML1.8 AND %ML7.24 THEN %WW3 := 0; END_IF;
(* Rung L51 *)
%QX1.7.14 := (%QX1.6.0 AND ((%ML8.7 AND NOT %QX1.6.6) OR (%ML8.8 AND %QX1.6.6))) OR (%QX1.6.0 AND %QX1.6.2 AND (%ML1.8 OR %QX1.7.14) AND NOT %ML0.14);
(* Rung L55 *)
%QX2.6.41 := (%QX1.6.0 AND %QX1.7.14) OR %ML101.0;
(* **********     HLV 20601선택 TK 104     ********** *)
(* Rung L58 *)
HLV_TK104_PANEL(CLK := %QX1.6.0 AND %QX1.6.3 AND %IX1.2.16);
%ML8.10 := HLV_TK104_PANEL.Q AND %QX1.6.3;
(* Rung L60 *)
IF %QX1.6.0 AND %QX1.6.2 AND %QX1.6.6 AND %ML1.9 AND %ML7.24 THEN %WW4 := 104; END_IF;
IF %QX1.6.0 AND %QX1.6.2 AND %QX1.6.6 THEN _t4 := %WW4 = 104; END_IF;
%ML8.11 := _t4;
(* Rung L67 *)
IF %QX1.6.0 AND NOT %ML1.9 AND %ML7.24 THEN %WW4 := 0; END_IF;

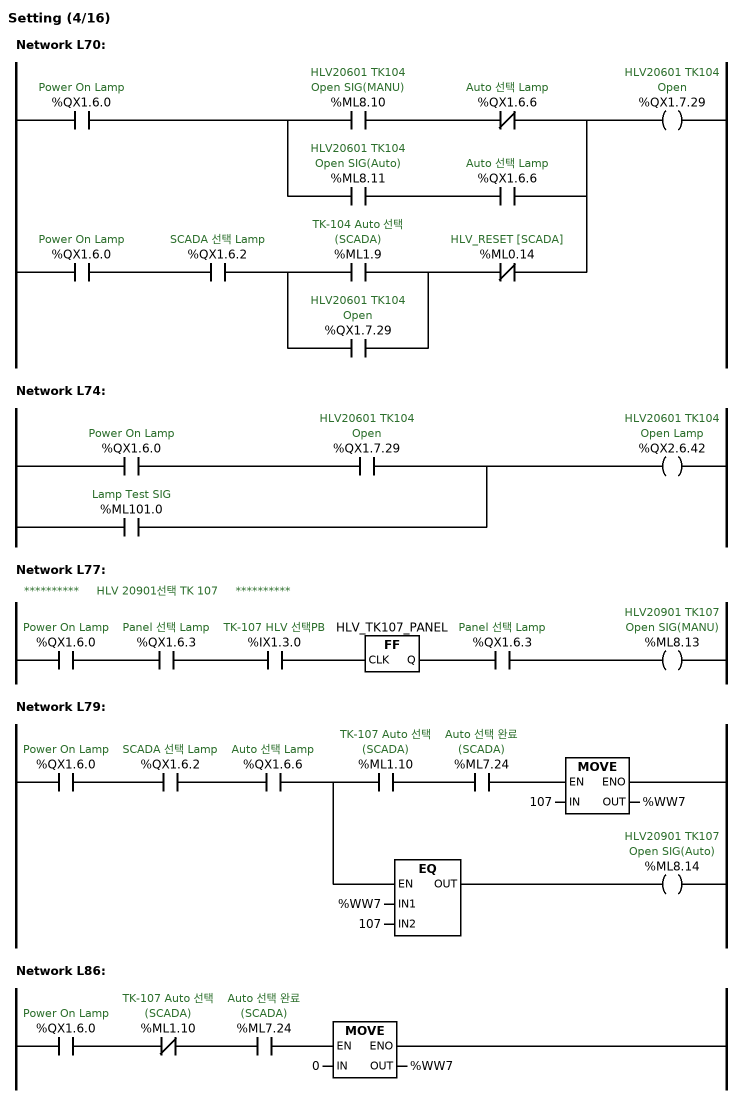
(* Rung L70 *)
%QX1.7.29 := (%QX1.6.0 AND ((%ML8.10 AND NOT %QX1.6.6) OR (%ML8.11 AND %QX1.6.6))) OR (%QX1.6.0 AND %QX1.6.2 AND (%ML1.9 OR %QX1.7.29) AND NOT %ML0.14);
(* Rung L74 *)
%QX2.6.42 := (%QX1.6.0 AND %QX1.7.29) OR %ML101.0;
(* **********     HLV 20901선택 TK 107     ********** *)
(* Rung L77 *)
HLV_TK107_PANEL(CLK := %QX1.6.0 AND %QX1.6.3 AND %IX1.3.0);
%ML8.13 := HLV_TK107_PANEL.Q AND %QX1.6.3;
(* Rung L79 *)
IF %QX1.6.0 AND %QX1.6.2 AND %QX1.6.6 AND %ML1.10 AND %ML7.24 THEN %WW7 := 107; END_IF;
IF %QX1.6.0 AND %QX1.6.2 AND %QX1.6.6 THEN _t5 := %WW7 = 107; END_IF;
%ML8.14 := _t5;
(* Rung L86 *)
IF %QX1.6.0 AND NOT %ML1.10 AND %ML7.24 THEN %WW7 := 0; END_IF;

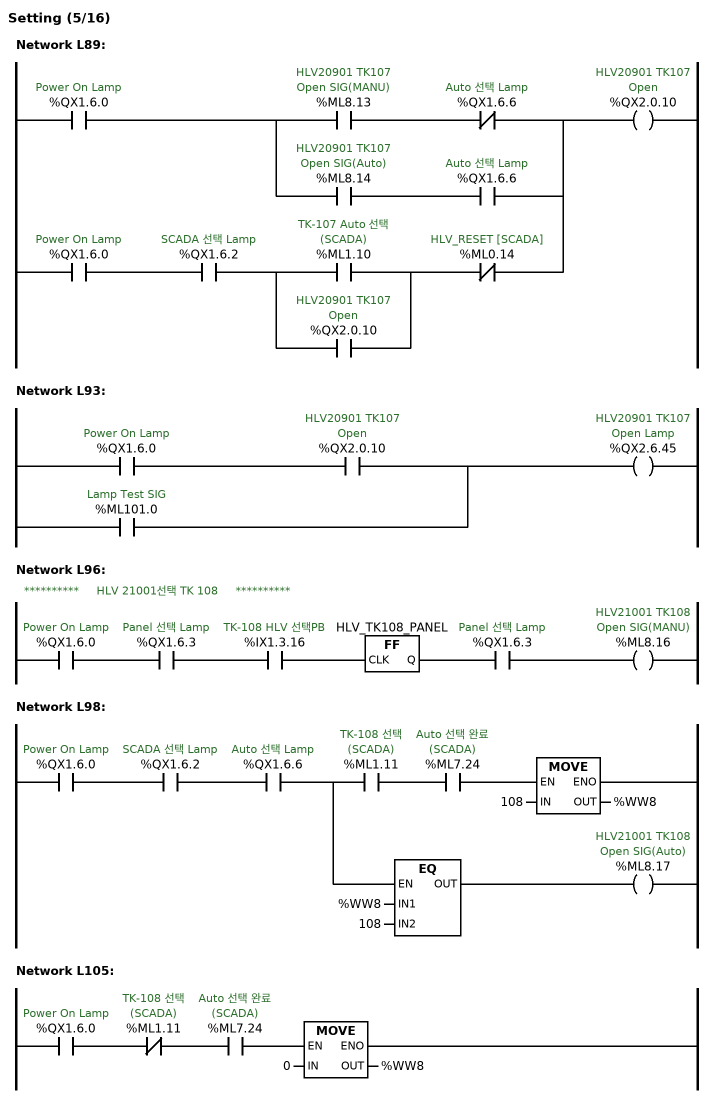
(* Rung L89 *)
%QX2.0.10 := (%QX1.6.0 AND ((%ML8.13 AND NOT %QX1.6.6) OR (%ML8.14 AND %QX1.6.6))) OR (%QX1.6.0 AND %QX1.6.2 AND (%ML1.10 OR %QX2.0.10) AND NOT %ML0.14);
(* Rung L93 *)
%QX2.6.45 := (%QX1.6.0 AND %QX2.0.10) OR %ML101.0;
(* **********     HLV 21001선택 TK 108     ********** *)
(* Rung L96 *)
HLV_TK108_PANEL(CLK := %QX1.6.0 AND %QX1.6.3 AND %IX1.3.16);
%ML8.16 := HLV_TK108_PANEL.Q AND %QX1.6.3;
(* Rung L98 *)
IF %QX1.6.0 AND %QX1.6.2 AND %QX1.6.6 AND %ML1.11 AND %ML7.24 THEN %WW8 := 108; END_IF;
IF %QX1.6.0 AND %QX1.6.2 AND %QX1.6.6 THEN _t6 := %WW8 = 108; END_IF;
%ML8.17 := _t6;
(* Rung L105 *)
IF %QX1.6.0 AND NOT %ML1.11 AND %ML7.24 THEN %WW8 := 0; END_IF;

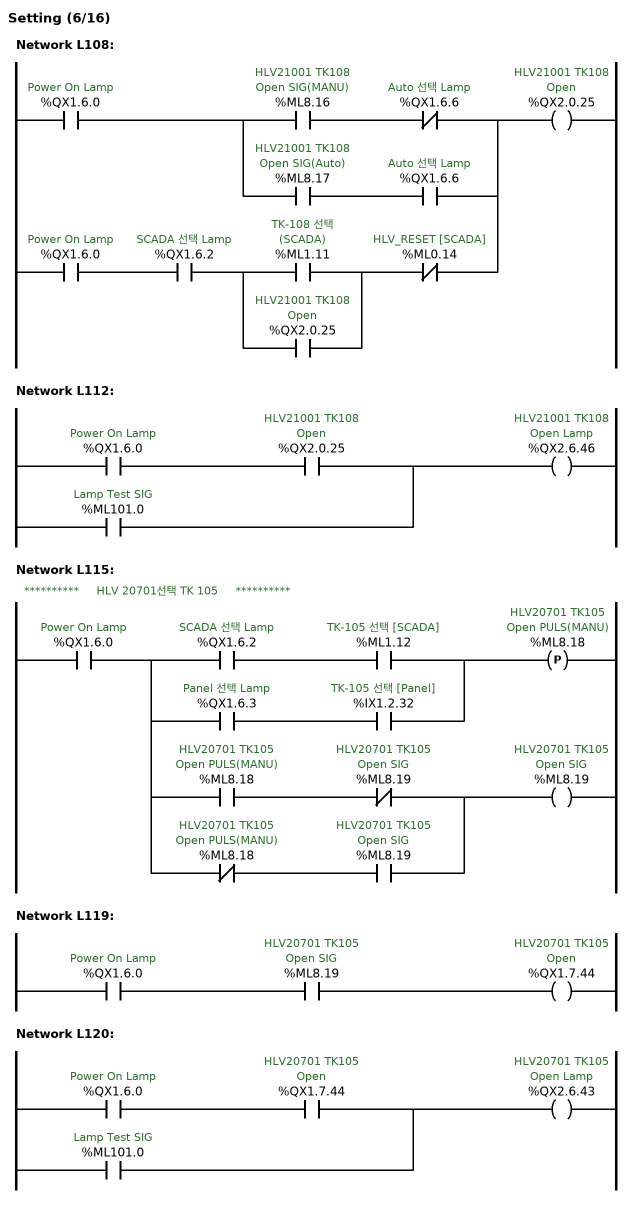
(* Rung L108 *)
%QX2.0.25 := (%QX1.6.0 AND ((%ML8.16 AND NOT %QX1.6.6) OR (%ML8.17 AND %QX1.6.6))) OR (%QX1.6.0 AND %QX1.6.2 AND (%ML1.11 OR %QX2.0.25) AND NOT %ML0.14);
(* Rung L112 *)
%QX2.6.46 := (%QX1.6.0 AND %QX2.0.25) OR %ML101.0;
(* **********     HLV 20701선택 TK 105     ********** *)
(* Rung L115 *)
_e7(CLK := %QX1.6.0 AND ((%QX1.6.2 AND %ML1.12) OR (%QX1.6.3 AND %IX1.2.32)));
%ML8.18 := _e7.Q;
%ML8.19 := %QX1.6.0 AND ((%ML8.18 AND NOT %ML8.19) OR (NOT %ML8.18 AND %ML8.19));
(* Rung L119 *)
%QX1.7.44 := %QX1.6.0 AND %ML8.19;
(* Rung L120 *)
%QX2.6.43 := (%QX1.6.0 AND %QX1.7.44) OR %ML101.0;

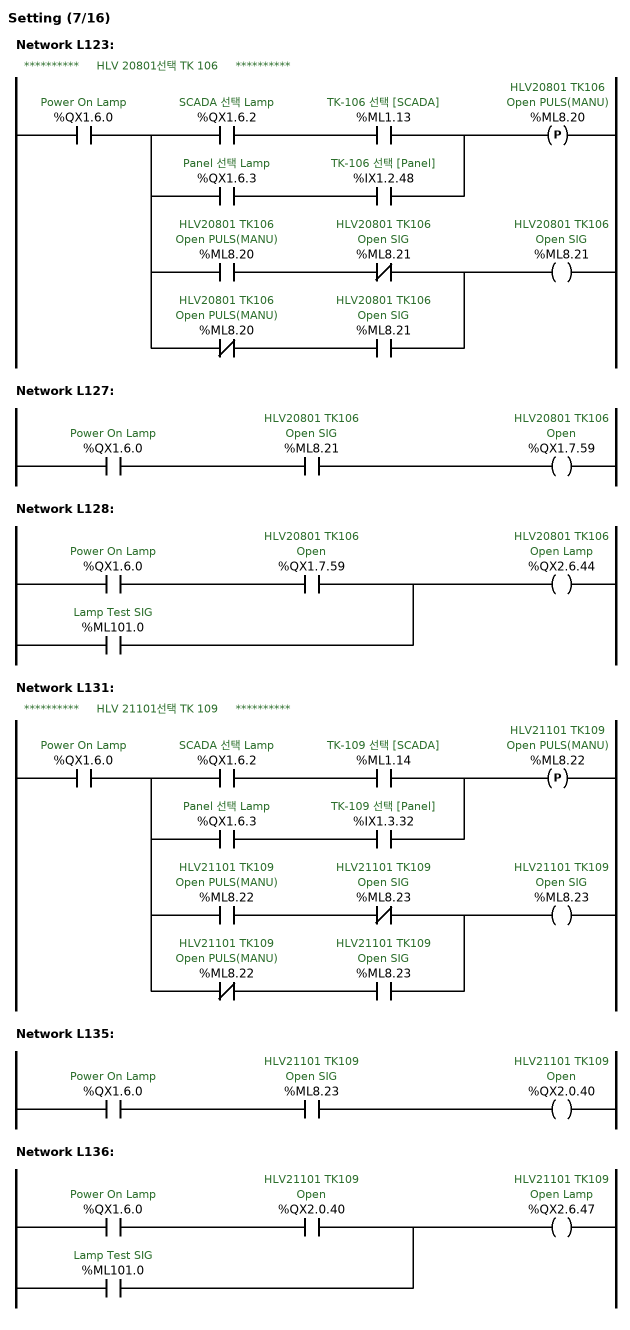
(* **********     HLV 20801선택 TK 106     ********** *)
(* Rung L123 *)
_e8(CLK := %QX1.6.0 AND ((%QX1.6.2 AND %ML1.13) OR (%QX1.6.3 AND %IX1.2.48)));
%ML8.20 := _e8.Q;
%ML8.21 := %QX1.6.0 AND ((%ML8.20 AND NOT %ML8.21) OR (NOT %ML8.20 AND %ML8.21));
(* Rung L127 *)
%QX1.7.59 := %QX1.6.0 AND %ML8.21;
(* Rung L128 *)
%QX2.6.44 := (%QX1.6.0 AND %QX1.7.59) OR %ML101.0;
(* **********     HLV 21101선택 TK 109     ********** *)
(* Rung L131 *)
_e9(CLK := %QX1.6.0 AND ((%QX1.6.2 AND %ML1.14) OR (%QX1.6.3 AND %IX1.3.32)));
%ML8.22 := _e9.Q;
%ML8.23 := %QX1.6.0 AND ((%ML8.22 AND NOT %ML8.23) OR (NOT %ML8.22 AND %ML8.23));
(* Rung L135 *)
%QX2.0.40 := %QX1.6.0 AND %ML8.23;
(* Rung L136 *)
%QX2.6.47 := (%QX1.6.0 AND %QX2.0.40) OR %ML101.0;

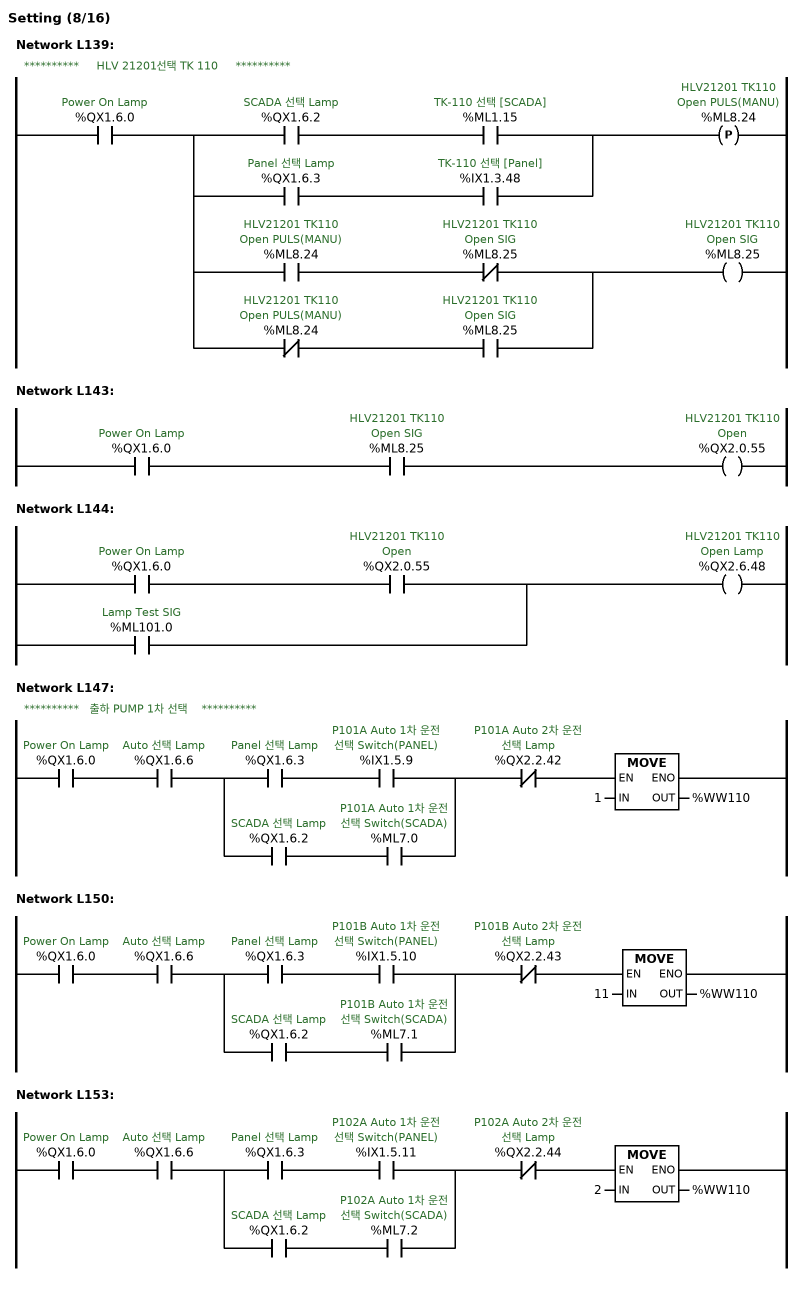
(* **********     HLV 21201선택 TK 110     ********** *)
(* Rung L139 *)
_e10(CLK := %QX1.6.0 AND ((%QX1.6.2 AND %ML1.15) OR (%QX1.6.3 AND %IX1.3.48)));
%ML8.24 := _e10.Q;
%ML8.25 := %QX1.6.0 AND ((%ML8.24 AND NOT %ML8.25) OR (NOT %ML8.24 AND %ML8.25));
(* Rung L143 *)
%QX2.0.55 := %QX1.6.0 AND %ML8.25;
(* Rung L144 *)
%QX2.6.48 := (%QX1.6.0 AND %QX2.0.55) OR %ML101.0;
(* **********   출하 PUMP 1차 선택    ********** *)
(* Rung L147 *)
IF %QX1.6.0 AND %QX1.6.6 AND ((%QX1.6.3 AND %IX1.5.9) OR (%QX1.6.2 AND %ML7.0)) AND NOT %QX2.2.42 THEN
    %WW110 := 1;
END_IF;
(* Rung L150 *)
IF %QX1.6.0 AND %QX1.6.6 AND ((%QX1.6.3 AND %IX1.5.10) OR (%QX1.6.2 AND %ML7.1)) AND NOT %QX2.2.43 THEN
    %WW110 := 11;
END_IF;
(* Rung L153 *)
IF %QX1.6.0 AND %QX1.6.6 AND ((%QX1.6.3 AND %IX1.5.11) OR (%QX1.6.2 AND %ML7.2)) AND NOT %QX2.2.44 THEN
    %WW110 := 2;
END_IF;

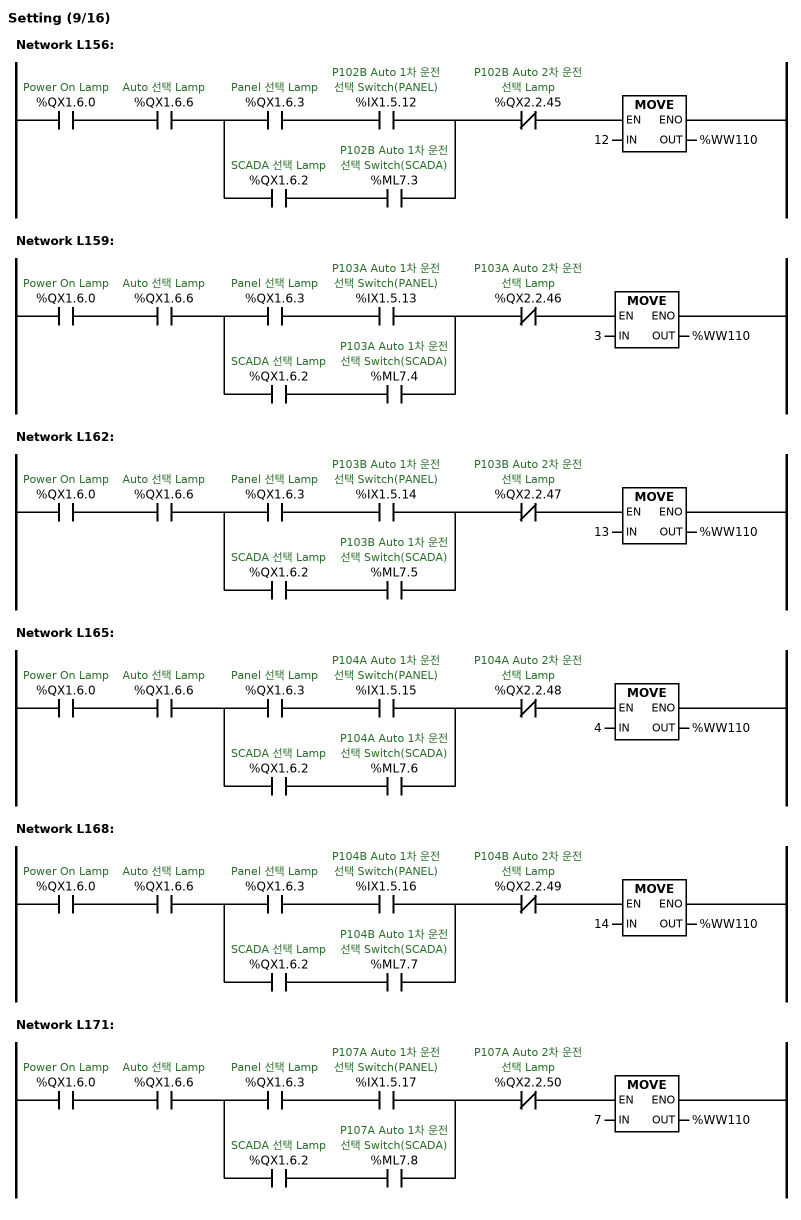
(* Rung L156 *)
IF %QX1.6.0 AND %QX1.6.6 AND ((%QX1.6.3 AND %IX1.5.12) OR (%QX1.6.2 AND %ML7.3)) AND NOT %QX2.2.45 THEN
    %WW110 := 12;
END_IF;
(* Rung L159 *)
IF %QX1.6.0 AND %QX1.6.6 AND ((%QX1.6.3 AND %IX1.5.13) OR (%QX1.6.2 AND %ML7.4)) AND NOT %QX2.2.46 THEN
    %WW110 := 3;
END_IF;
(* Rung L162 *)
IF %QX1.6.0 AND %QX1.6.6 AND ((%QX1.6.3 AND %IX1.5.14) OR (%QX1.6.2 AND %ML7.5)) AND NOT %QX2.2.47 THEN
    %WW110 := 13;
END_IF;
(* Rung L165 *)
IF %QX1.6.0 AND %QX1.6.6 AND ((%QX1.6.3 AND %IX1.5.15) OR (%QX1.6.2 AND %ML7.6)) AND NOT %QX2.2.48 THEN
    %WW110 := 4;
END_IF;
(* Rung L168 *)
IF %QX1.6.0 AND %QX1.6.6 AND ((%QX1.6.3 AND %IX1.5.16) OR (%QX1.6.2 AND %ML7.7)) AND NOT %QX2.2.49 THEN
    %WW110 := 14;
END_IF;
(* Rung L171 *)
IF %QX1.6.0 AND %QX1.6.6 AND ((%QX1.6.3 AND %IX1.5.17) OR (%QX1.6.2 AND %ML7.8)) AND NOT %QX2.2.50 THEN
    %WW110 := 7;
END_IF;

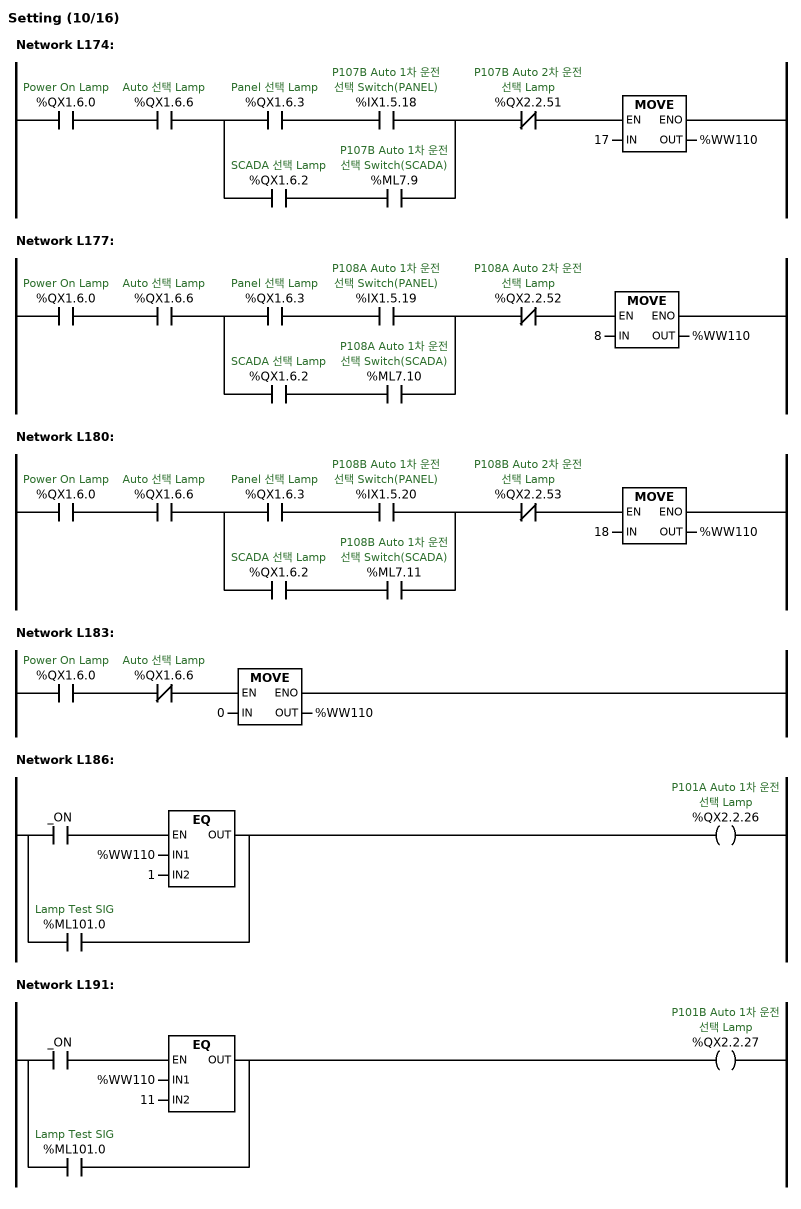
(* Rung L174 *)
IF %QX1.6.0 AND %QX1.6.6 AND ((%QX1.6.3 AND %IX1.5.18) OR (%QX1.6.2 AND %ML7.9)) AND NOT %QX2.2.51 THEN
    %WW110 := 17;
END_IF;
(* Rung L177 *)
IF %QX1.6.0 AND %QX1.6.6 AND ((%QX1.6.3 AND %IX1.5.19) OR (%QX1.6.2 AND %ML7.10)) AND NOT %QX2.2.52 THEN
    %WW110 := 8;
END_IF;
(* Rung L180 *)
IF %QX1.6.0 AND %QX1.6.6 AND ((%QX1.6.3 AND %IX1.5.20) OR (%QX1.6.2 AND %ML7.11)) AND NOT %QX2.2.53 THEN
    %WW110 := 18;
END_IF;
(* Rung L183 *)
IF %QX1.6.0 AND NOT %QX1.6.6 THEN %WW110 := 0; END_IF;
(* Rung L186 *)
IF _ON THEN _t11 := %WW110 = 1; END_IF;
%QX2.2.26 := _t11 OR %ML101.0;
(* Rung L191 *)
IF _ON THEN _t12 := %WW110 = 11; END_IF;
%QX2.2.27 := _t12 OR %ML101.0;

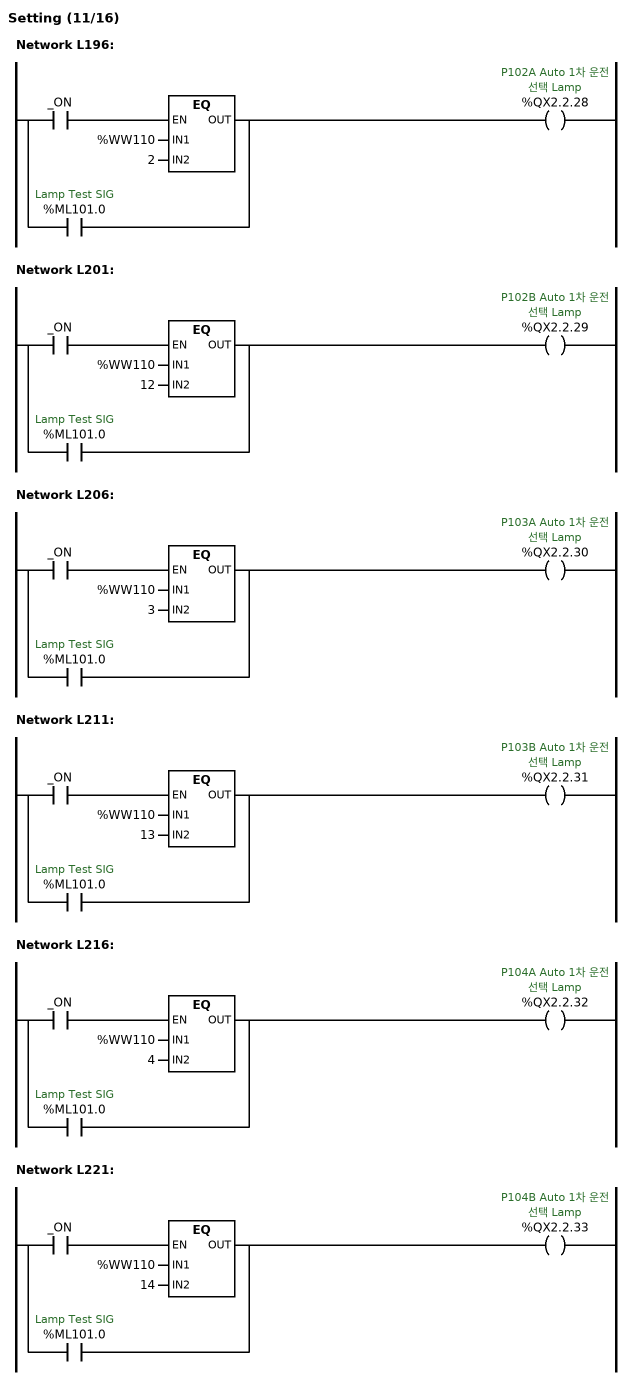
(* Rung L196 *)
IF _ON THEN _t13 := %WW110 = 2; END_IF;
%QX2.2.28 := _t13 OR %ML101.0;
(* Rung L201 *)
IF _ON THEN _t14 := %WW110 = 12; END_IF;
%QX2.2.29 := _t14 OR %ML101.0;
(* Rung L206 *)
IF _ON THEN _t15 := %WW110 = 3; END_IF;
%QX2.2.30 := _t15 OR %ML101.0;
(* Rung L211 *)
IF _ON THEN _t16 := %WW110 = 13; END_IF;
%QX2.2.31 := _t16 OR %ML101.0;
(* Rung L216 *)
IF _ON THEN _t17 := %WW110 = 4; END_IF;
%QX2.2.32 := _t17 OR %ML101.0;
(* Rung L221 *)
IF _ON THEN _t18 := %WW110 = 14; END_IF;
%QX2.2.33 := _t18 OR %ML101.0;

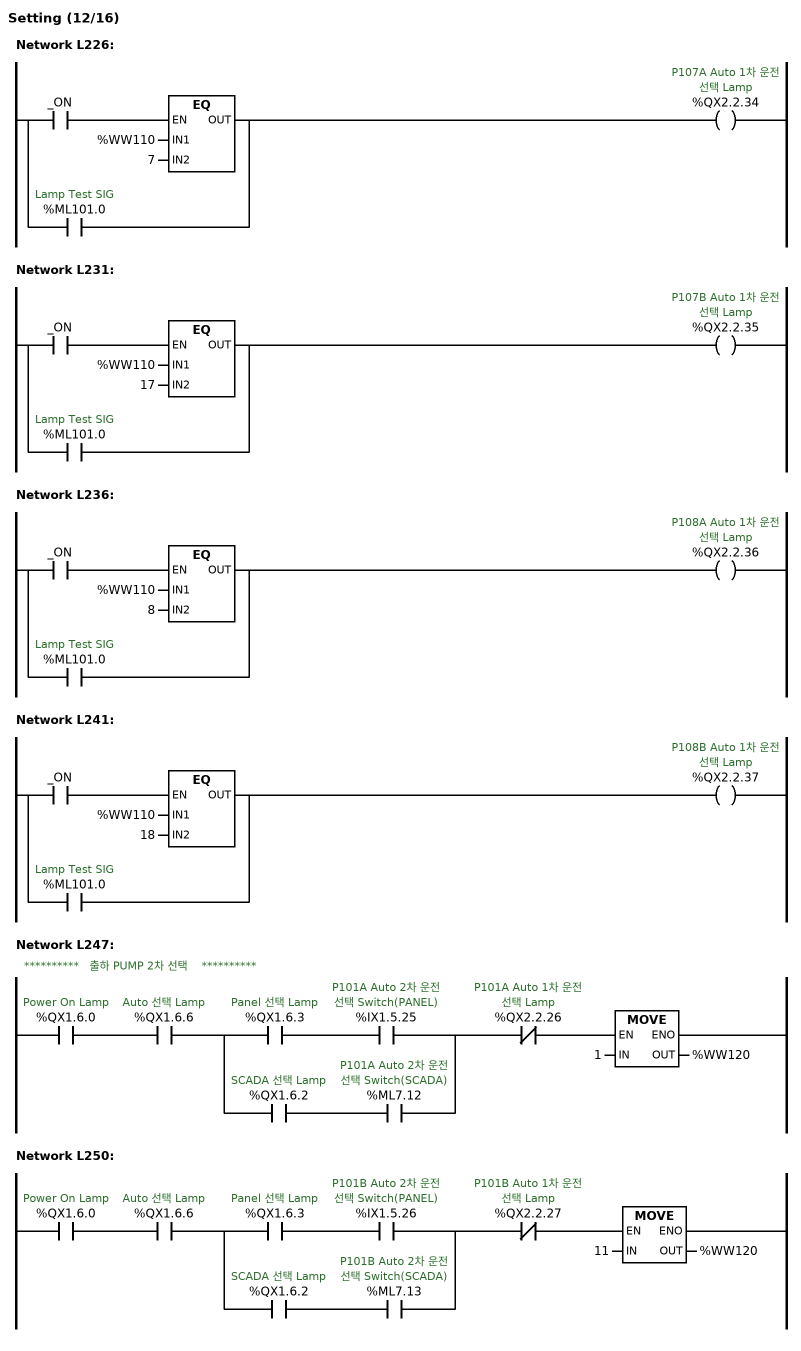
(* Rung L226 *)
IF _ON THEN _t19 := %WW110 = 7; END_IF;
%QX2.2.34 := _t19 OR %ML101.0;
(* Rung L231 *)
IF _ON THEN _t20 := %WW110 = 17; END_IF;
%QX2.2.35 := _t20 OR %ML101.0;
(* Rung L236 *)
IF _ON THEN _t21 := %WW110 = 8; END_IF;
%QX2.2.36 := _t21 OR %ML101.0;
(* Rung L241 *)
IF _ON THEN _t22 := %WW110 = 18; END_IF;
%QX2.2.37 := _t22 OR %ML101.0;
(* **********   출하 PUMP 2차 선택    ********** *)
(* Rung L247 *)
IF %QX1.6.0 AND %QX1.6.6 AND ((%QX1.6.3 AND %IX1.5.25) OR (%QX1.6.2 AND %ML7.12)) AND NOT %QX2.2.26 THEN
    %WW120 := 1;
END_IF;
(* Rung L250 *)
IF %QX1.6.0 AND %QX1.6.6 AND ((%QX1.6.3 AND %IX1.5.26) OR (%QX1.6.2 AND %ML7.13)) AND NOT %QX2.2.27 THEN
    %WW120 := 11;
END_IF;

